FUNCTION_BLOCK "FB_HUB_FW_re"   // FB23, STL
{ S7_Optimized_Access := 'FALSE' }
AUTHOR : MS
// stored: AutoNumber false
   VAR_INPUT
      FW_DBNr : Int;
      SysTime : Time;
   END_VAR
   VAR
      Config : Struct
         Speed : Struct
            Min : Int;   // Mindestgeschwindigkeit in %
            Tipp : Int;   // Geschwindigkeit bei Tipp-Betrieb in %
            Hand : Int;   // maximale Geschwindigkeit bei Hand-Betrieb in %
            Max : Int;   // maximale Geschwindigkeit bei Automatik-Betrieb in %
            Norm : Real;   // Geschwindigkeit in INC/s bei 100%
            endMess : Real;   // gemessene Geschwindigkeit in INC/s bei 100%
         END_STRUCT;
         Rampe : Struct
            Auf_Heben : Real;   // Zeit für Beschleunigung beim Heben von 0% auf 200%
            Ab_Heben : Real;   // Zeit für Verzögerung bei Heben von 200% auf 0%
            Auf_Senken : Real;   // Zeit für Beschleunigung bei Senken von 0% auf 200%
            Ab_Senken : Real;   // Zeit für Verzögerung bei Senken von 200% auf 0%
            NotStop : Real;   // Zeit für Verzögerung bei NotStopp von 200% auf 0%
         END_STRUCT;
         Bereich : Struct
            Pos : DInt;
            Stop : DInt;
            Ziel : DInt;
            Absetzen : DInt;
            Langsam : DInt;
         END_STRUCT;
         TV_Position : DInt;   // Verzögerung Ebenenmitte in ms
         Reaktionszeit : Int;   // Reaktionszeit FU
         Startzeit : Int;   // Zeit Startverzögerung in ms (Zeit von erster Sollwertausgabe bis Istwert>0)
         Variante : Byte;   // Art der Positionierung (0-Absolut, 1-SensorSys, 2-..)
         SimIstSpeed : Byte;   // Variante Simulation Istgeschwindigkeit (0-aus, 1-Soll=Ist,...)
         SimSensors : DWord := DWORD#16#4400_0022;   // Sensoraufbau für Simulation
         SimTakt : DInt;   // Schiebetakt für Sensorsimu in ms
      END_STRUCT;
      IN : Struct
         BA_Tipp : Bool;   // Betriebsart FW Tipp
         BA_Hand : Bool;   // Betriebsart FW Hand
         BA_Auto : Bool;   // Betriebsart FW Auto
         Heben_aktiv : Bool;
         Frg_Hub : Bool;   // Freigabe Positioniervorgang
         Frg_Eil : Bool;   // max. Speed in Automatik und Hand-Speed in Tipp erlaubt
         Break_on : Bool;   // Rückmeldung extern Bremse eingefallen / Hubwerk steht
         mittig : Bool;   // Hub in Posmitte
         resB : Byte;
         HubInc : DInt;   // Istposition in Inkrementen (mm)
         ZielInc : DInt;   // Ziel in Inkrenmenten (mm)
         Absetz_Inc : DInt;   // Inkrement der SU-Ebene des FW
         IstSpeed : Int;   // Istgeschwindigkeit in %
      END_STRUCT;
      OUT : Struct
         Hub_Ok : Bool;   // Positionierung beendet FW steht
         Break_off : Bool;   // Bremse lösen
         res_1 : Bool;
         res_2 : Bool;
         res_3 : Bool;
         res_4 : Bool;
         res_5 : Bool;
         res_6 : Bool;
         resB : Byte;
         Bereich_langsam : DInt;   // berechneter Anhaltebereich
         SollSpeed : Int;   // Sollgeschwindigkeit in %
      END_STRUCT;
      Tmp : Struct
         lastTime : DInt;   // letzter Systemzeitpunkt
         DiffTime : Real;   // Zeit seit letzter Bearbeitung
         lastSpeed : Real;   // letzte ausgegebene Geschwindigkeit
         Messung : Struct
            lastInc : Real;
            addInc : Real;
            addTime : Real;
            lastIst : Int;
            messAct : Bool;
         END_STRUCT;
         StopCount : DInt;
         subInc : Real;
         lastOut : Real;
         TaktCount : Real;   // Taktzähler für Sensorsimu
         PtrSensors : DWord := DWORD#16#0000_0001;
         RunTime : DInt;   // Zeit seit Start Positioniervorgang
      END_STRUCT;
   END_VAR
   VAR_TEMP
      FWDB : Int;
      Rampe_Auf : Real;
      Rampe_Ab : Real;
      minSpeed : Real;
      maxSpeed : Real;
      normSpeed : Real;
      handSpeed : Real;
      TippSpeed : Real;
      IstSpeed : Real;
      Abstand : Real;
      maxDelta : Real;
      Speed : Real;
      tx : Real;
      Rampe_Not : Real;
      incDelta : DInt;
      messAct : Bool;
      posAbsolut : Bool;
      Sensor_on : Bool;
      no_Brms : Bool;
      savD_1 : DInt;
      savD_2 : DInt;
      Korrmax : Real;   // Korrektur max-Speed vom WT
   END_VAR
BEGIN

NETWORK
TITLE = Daten aus FW lesen

      L     #FW_DBNr;
      T     #FWDB;
      OPN   DB [#FWDB];
      AN    "DI_FW_1".IN.Com_Reset;
      JC    nRes;
      L     #SysTime;
      T     #Tmp.lastTime;
      L     0.0;
      T     #Tmp.lastSpeed;
      T     #Tmp.subInc;

nRes: A     "DI_FW_1".ZST.Auto;
      =     #IN.BA_Auto;
      A     "DI_FW_1".ZST.Hand;
      =     #IN.BA_Hand;
      A     "DI_FW_1".ZST.Tipp;
      O     "DI_FW_1".OUT.TIPP;
      =     #IN.BA_Tipp;
      R     #IN.BA_Auto;
      R     #IN.BA_Hand;

      A     "DI_FW_1".OUT.HEBEN_re;
      =     #IN.Heben_aktiv;

      A     "DI_FW_1".OUT.HEBEN_re;
      O     "DI_FW_1".OUT.SENKEN_re;
      =     #IN.Frg_Hub;

      A     "DI_FW_1".OUT.HUB_EIL_re;
      =     #IN.Frg_Eil;

      A     "DI_FW_1".ZST.Mittig;
      =     #IN.mittig;

      A     "DI_FW_1".OUT.no_Brms;
      =     #no_Brms;

      L     "DI_FW_1".HELP.HubInc_re;
      T     #IN.HubInc;
      L     "DI_FW_1".HELP.HubZielInc_re;
      T     #IN.ZielInc;

      L     "DI_FW_1".TMP.low_SU_Ebene;
      L     4;
      *D;
      L     292;
      +D;
      SLD   3;
      LAR1;
      OPN   DB [#FWDB];
      L     DBD [AR1, P#0.0];  //"DI_FW_1".PAR.Hub.Ebene0
      L     #Config.Bereich.Absetzen;
      +D;
      T     #IN.Absetz_Inc;

      L     "DI_FW_1".PAR.Hub.WT_Speed;
      ITD;
      DTR;
      L     100.0;
      /R;
      L     #Config.Speed.Max;
      ITD;
      DTR;
      *R;
      T     #Korrmax;


NETWORK
TITLE = kein Auftrag/Initialisieren
//----------------------------------------
//Positionierart
//----------------------------------------
      L     #Config.Variante;
      L     0;
      ==I;
      =     #posAbsolut;

//----------------------------------------
//Zeitmessung
//----------------------------------------
      L     #SysTime;
      L     #Tmp.lastTime;
      >=D;
      JC    nUms;
      L     16#7FFF_FFFF;  //L#2147483647
      CAC;
      -D;
      L     #SysTime;
      +D;
      JU    Ums;
nUms: -D;
Ums:  DTR;
      T     #Tmp.DiffTime;
      L     10.0;  //Berechnung unter 10ms zu ungenau
      <R;
      BEC;

      L     #SysTime;
      T     #Tmp.lastTime;

//----------------------------------------
//Parametersatz laden
//----------------------------------------
// :::::::::::::::::::::::::::::::::::::::
// Rampen
// :::::::::::::::::::::::::::::::::::::::
      A     #IN.Heben_aktiv;
      O     #IN.BA_Tipp;
      L     #Config.Rampe.Auf_Heben;
      JC    slu;
      L     #Config.Rampe.Auf_Senken;
slu:  L     1000.0;
      *R;
      L     2.0;
      /R;
      T     #Rampe_Auf;

      A     #IN.Heben_aktiv;
      O     #IN.BA_Tipp;
      L     #Config.Rampe.Ab_Heben;
      JC    sld;
      L     #Config.Rampe.Ab_Senken;
sld:  L     1000.0;
      *R;
      L     2.0;
      /R;
      T     #Rampe_Ab;

// :::::::::::::::::::::::::::::::::::::::
// Normalgeschwindigkeit
// :::::::::::::::::::::::::::::::::::::::
      L     #Config.Speed.Norm;
      L     1000.0;
      /R;
      T     #normSpeed;

// :::::::::::::::::::::::::::::::::::::::
// Istgeschwindigkeit
// :::::::::::::::::::::::::::::::::::::::
      L     #IN.IstSpeed;
      ITD;
      DTR;
      ABS;
      L     10000.0;
      /R;
      L     #normSpeed;
      *R;
      T     #IstSpeed;

// :::::::::::::::::::::::::::::::::::::::
// Abstand
// :::::::::::::::::::::::::::::::::::::::
      L     #IN.HubInc;
      L     #IN.ZielInc;
      -D;
      DTR;
      ABS;
      T     #Abstand;

//Korrektur Abstand (Vorhalteweg)um Reaktionszeit auszugleichen
      AN    #posAbsolut;
      JC    StA;
      L     #Config.Reaktionszeit;  //VorhalteWeg=Istspeed * Reaktionszeit
      ITD;  //s = v*t
      DTR;
      L     #IstSpeed;
      *R;
      L     #Abstand;
      CAC;
      -R;
      L     0.0;
      <=R;
      JC    StA;
      CAC;
StA:  T     #Abstand;


// :::::::::::::::::::::::::::::::::::::::
// --- Geschwindigkeiten (Min, Hand, Max)
// :::::::::::::::::::::::::::::::::::::::
      L     #Config.Speed.Tipp;
      A     #IN.BA_Tipp;
      JC    min;
      L     #Config.Speed.Min;
min:  DTR;
      ABS;
      L     100.0;
      /R;
      L     #normSpeed;
      *R;
      T     #minSpeed;

      L     #Config.Speed.Hand;
      DTR;
      ABS;
      L     100.0;
      /R;
      L     #normSpeed;
      *R;
      T     #handSpeed;

      L     #Config.Speed.Tipp;
      DTR;
      ABS;
      L     100.0;
      /R;
      L     #normSpeed;
      *R;
      T     #TippSpeed;

// 2021-07-09 Heben /Senken gleich
      L     #IN.HubInc;
      L     #IN.Absetz_Inc;
      <=D;
      AN    #IN.Frg_Eil;
      A     #IN.mittig;  // Korb am Haken
      O     #IN.BA_Tipp;
      L     #Config.Speed.Tipp;
      JC    max;

      AN    #IN.mittig;
      L     #Config.Speed.Max;  // Höhenwechsel + Freifahren
      JC    max;

      L     #IN.HubInc;
      L     #IN.Absetz_Inc;
      <=D;
      L     #Config.Speed.Hand;
      PUSH;
      +D;
      JC    max;
//
      L     #Config.Speed.Max;
max:  DTR;
      ABS;
      L     #Korrmax;
      >R;
      JC    korr;
      CAC;
korr: L     100.0;
      /R;
      L     #normSpeed;
      *R;
      T     #maxSpeed;
      L     #minSpeed;
      >=R;
      JC    okmx;
      T     #maxSpeed;

//----------------------------------------
//kein Auftrag
//----------------------------------------
okmx: AN    #IN.Frg_Hub;
      JC    Off;

      L     #Tmp.DiffTime;
      L     #Tmp.RunTime;
      +R;
      T     #Tmp.RunTime;

      AN    #IN.BA_Tipp;
      JC    Auto;


NETWORK
TITLE = Tipp
      A     #IN.Frg_Eil;
      L     #maxSpeed;
      JC    Tout;
      L     #minSpeed;
Tout: T     #Speed;
      JU    OutW;

NETWORK
TITLE = Positioniervariante aussuchen
Auto: SET;
      R     #OUT.Hub_Ok;

      L     #Config.Variante;
      JL    vErr;
      JU    vAbs;  //0 Absolut direkt
      JU    vSen;  //1 mit Sensor-System
vErr: JU    Off;


NETWORK
TITLE = Positionierung Absolut direkt
vAbs: NOP   0;

//----------------------------------------
// Bereich_Langsam berechnen
//
// s = (Rampe * Vist * Vist) / (2 * Vnorm)
//----------------------------------------
      L     #Rampe_Ab;
      L     0.0;
      <=R;
      L     #Config.Bereich.Langsam;
      JC    setB;

      L     #IstSpeed;
      SQR;
      L     #Rampe_Ab;
      *R;
      L     #normSpeed;
      /R;
      L     2.0;
      /R;
      RND;
setB: T     #OUT.Bereich_langsam;

//----------------------------------------
// maximal mögl. Geschwindigkeit berechnen
//
// v = SQRT(2 * s * Vnorm / Rampe)
//----------------------------------------
      L     #Abstand;
      L     #Config.Bereich.Ziel;
      DTR;
      >R;
      JC    Sped;

      L     #Abstand;
      L     #Config.Bereich.Stop;
      DTR;
      >R;
      L     #minSpeed;
      JC    setS;

      L     0;
      JU    setS;

Sped: L     #Rampe_Ab;
      L     0.0;
      <=R;
      L     #maxSpeed;
      JC    setS;

      L     2.0;
      L     #Abstand;
      *R;
      L     #normSpeed;
      *R;
      L     #Rampe_Ab;
      /R;
      SQRT;
setS: T     #Speed;

//----------------------------------------
// MAX begrenzen beim Senken (Absetzen)
//
// Vmax = SQRT(2 * Abstand * V100 / t100 + Vhand * Vhand)
//----------------------------------------
      L     #Rampe_Ab;
      L     0.0;
      <=R;
      O     #IN.Heben_aktiv;
      JC    aMax;

      L     #IN.HubInc;
      L     #IN.Absetz_Inc;
      <=D;
      JC    aMax;

      L     #IN.HubInc;
      L     #IN.Absetz_Inc;
      -D;
      DTR;
      L     2.0;
      *R;
      L     #normSpeed;
      *R;
      L     #Rampe_Ab;
      /R;
      L     #handSpeed;
      SQR;
      +R;
      SQRT;
      L     #maxSpeed;
      >R;
      JC    aMax;
      CAC;
      T     #maxSpeed;

//----------------------------------------
// errechnete Geschwindigkeit auf MAX begrenzen
//----------------------------------------
aMax: L     #Speed;
      L     #maxSpeed;
      <=R;
      JC    Ramp;
      T     #Speed;
      JU    Ramp;

//----------------------------------------
// Anstiegsrampe begrenzen
//
// Vdelta = (Vnorm * Tdelta / Rampe)
//----------------------------------------
Ramp: L     #Speed;
      L     #IstSpeed;
      <=R;
      JC    aMin;

      L     #Rampe_Auf;
      L     0.0;
      <=R;
      JC    aMin;

      L     #Tmp.RunTime;
      L     #Config.Startzeit;
      DTR;
      <R;
      L     #minSpeed;
      JC    altw;

      L     #normSpeed;
      L     #Tmp.DiffTime;
      *R;
      L     #Rampe_Auf;
      /R;
      T     #maxDelta;

      L     #Speed;
      L     #Tmp.lastOut;
      -R;
      ABS;
      L     #maxDelta;
      <=R;
      JC    aMin;

      L     #Tmp.lastOut;
      +R;
altw: T     #Speed;

//----------------------------------------
// errechnete Geschwindigkeit auf MIN begrenzen
//----------------------------------------
aMin: L     #Speed;
      L     #minSpeed;
      >=R;
      JC    Out;

      T     #Speed;

      JU    Out;


NETWORK
TITLE = Positionierung mit Sensor-System
vSen: SET;
// -------------------------------
// Geschwindigkeit berechnen
// -------------------------------
      L     #Abstand;
      L     #Config.Bereich.Langsam;
      DTR;
      >R;
      L     #maxSpeed;
      JC    vSet;

      L     #Abstand;
      L     #Config.Bereich.Ziel;
      DTR;
      <=R;
      L     #minSpeed;
      JC    vSet;

      A     #no_Brms;
      L     #maxSpeed;
      JC    vSet;

      L     #handSpeed;
      L     #maxSpeed;
      >R;
      JC    vSet;
      CAC;

vSet: T     #Speed;

// -------------------------------
// Rampen begrenzen
// -------------------------------
      L     #Speed;
      L     #IstSpeed;
      >R;
      JC    rAuf;
      <R;
      JC    rAb;
      JU    Out;

rAuf: L     0.0;
      L     #Rampe_Auf;
      >=R;
      JC    Out;

      L     #Tmp.RunTime;
      L     #Config.Startzeit;
      DTR;
      >=R;
      JC    wtr2;

      L     #minSpeed;
      JU    outS;

wtr2: L     #normSpeed;
      L     #Tmp.DiffTime;
      *R;
      L     #Rampe_Auf;
      /R;
      T     #maxDelta;

      L     #Speed;
      L     #Tmp.lastOut;
      -R;
      ABS;
      L     #maxDelta;
      <=R;
      JC    Out;

      L     #Tmp.lastOut;
      +R;
outS: T     #Speed;
      JU    Out;

rAb:  L     0.0;
      L     #Rampe_Ab;
      >=R;
      JC    Out;

      L     #normSpeed;
      L     #Tmp.DiffTime;
      *R;
      L     #Rampe_Ab;
      /R;
      T     #maxDelta;

      L     #Tmp.lastOut;
      L     #Speed;
      -R;
      ABS;
      L     #maxDelta;
      <=R;
      JC    Out;

      L     #Tmp.lastOut;
      CAC;
      -R;
      T     #Speed;
      JU    Out;


NETWORK
TITLE = Ausgabe
Out:  L     #Abstand;
      L     #Config.Bereich.Ziel;
      DTR;
      >R;
      L     #Config.TV_Position;
      DTR;
      JC    setT;

      L     #minSpeed;
      T     #Speed;

      L     #Tmp.StopCount;
      L     0.0;
      <=R;
      O(;
      L     #Abstand;
      L     #Config.Bereich.Stop;
      DTR;
      <=R;
      A     #posAbsolut;
      );
      JC    Off;

      L     #Tmp.StopCount;
      L     #Tmp.DiffTime;
      -R;

setT: T     #Tmp.StopCount;
      JU    OutW;

Off:  A     #IN.Break_on;
      S     #OUT.Hub_Ok;

      L     0;
      T     #OUT.Bereich_langsam;
      L     0.0;
      T     #Speed;
      T     #Tmp.lastOut;
      T     #Tmp.RunTime;
      JU    OutW;

OutW: L     #Speed;
      T     #Tmp.lastOut;
      L     100.0;
      *R;
      L     #normSpeed;
      /R;
      T     #maxDelta;
      TRUNC;
      T     #OUT.SollSpeed;

      L     #Tmp.RunTime;
      L     #Config.Startzeit;
      DTR;
      >=R;
      A     #IN.Frg_Hub;
      S     #OUT.Break_off;

      L     #OUT.SollSpeed;
      L     0;
      ==I;
      ON    #IN.Frg_Hub;
      R     #OUT.Break_off;


NETWORK
TITLE = Messung der Normgeschwindigkeit
      L     #IN.IstSpeed;
      L     #Tmp.Messung.lastIst;
      -I;
      JP    cNeg;
      NEGI;
cNeg: L     100;
      <=I;
      A     #IN.Frg_Hub;
      =     #messAct;
      JC    cOn;
//----------------------------------------
// Messung aus
// Werte initialisieren
//----------------------------------------
      L     0.0;
      T     #Tmp.Messung.addTime;
      T     #Tmp.Messung.addInc;

      L     #IN.IstSpeed;
      T     #Tmp.Messung.lastIst;
      JU    cEnd;

//----------------------------------------
// Messung läuft
// Werte aufzeichnen
//----------------------------------------
cOn:  L     #IN.HubInc;
      DTR;
      L     #Tmp.Messung.lastInc;
      -R;
      ABS;
      L     #Tmp.Messung.addInc;
      +R;
      T     #Tmp.Messung.addInc;

      L     #Tmp.DiffTime;
      L     #Tmp.Messung.addTime;
      +R;
      T     #Tmp.Messung.addTime;

//----------------------------------------
// Messung läuft lange genug
// um Werte zu berechnen
//----------------------------------------
      L     #Tmp.Messung.addTime;
      L     1000.0;
      <R;
      JC    cEnd;
      /R;
      L     #Tmp.Messung.addInc;
      CAC;
      /R;
      L     #Tmp.Messung.lastIst;
      ITD;
      DTR;
      ABS;
      /R;
      L     10000.0;
      *R;
      T     #Config.Speed.endMess;
      JU    cEnd;

cEnd: L     #IN.HubInc;
      DTR;
      T     #Tmp.Messung.lastInc;



NETWORK
TITLE = Daten in FW schreiben

      OPN   DB [#FWDB];

      A     #OUT.Hub_Ok;
      =     "DI_FW_1".IN.Hub_ok_re;

      L     #OUT.SollSpeed;
      T     "DI_FW_1".HELP.Speed_Hub_re;


NETWORK
TITLE = Simulation Ist-Wert-Rückgabe
      L     #Config.SimIstSpeed;
      L     0;
      ==I;
      JC    simu;

      L     #OUT.SollSpeed;
      T     #IN.IstSpeed;

simu: NOP   0;


NETWORK
TITLE = Simulation Bewegung
      AN    "DB_ANLAGE".BA.Simulation;
      BEC;

      AN    #OUT.Break_off;
      =     #IN.Break_on;

      A     #IN.Heben_aktiv;
      JC    sTra;
      L     #Speed;
      NEGR;
      T     #Speed;
sTra: L     #Config.Rampe.NotStop;
      L     0.0;
      <=R;
      JC    Ink;

      L     #Config.Rampe.NotStop;
      L     1000.0;
      *R;
      L     2.0;
      /R;
      T     #Rampe_Not;

      L     #normSpeed;
      L     #Tmp.DiffTime;
      *R;
      L     #Rampe_Not;
      /R;
      T     #maxDelta;

      L     #Speed;
      L     #Tmp.lastSpeed;
      -R;
      ABS;
      L     #maxDelta;
      <=R;
      JC    Ink;

      L     #Speed;
      L     #Tmp.lastSpeed;
      <R;
      L     #Tmp.lastSpeed;
      L     #maxDelta;
      JC    sub;
      +R;
      JU    stt;
sub:  -R;
stt:  T     #Speed;

Ink:  L     #Config.Variante;
      JL    sErr;
      JU    sAbs;  //0 Absolut direkt
      JU    sSen;  //1 mit Sensor-System
sErr: JU    OutS_Mig;

//----------------------------------------
// Simu Absolut
//----------------------------------------
sAbs: L     #Speed;
      L     #Tmp.lastSpeed;
      +R;
      L     2.0;
      /R;
      L     #Tmp.DiffTime;
      *R;
      L     #Tmp.subInc;
      +R;
      T     #Tmp.subInc;

      TRUNC;
      T     #incDelta;
      L     #IN.HubInc;  // init startinkrement
      +D;
      OPN   DB [#FWDB];
      T     "DI_FW_1".HELP.HubInc_re;

      L     #Tmp.subInc;
      L     #incDelta;
      DTR;
      -R;
      T     #Tmp.subInc;
      JU    OutS_Mig;

//------------------------------------------
// Simu Sensoren
//------------------------------------------

// :::::::::::::::::::::::::::::::::::::::::
// Simulationstakt entsprechend IstSpeed
// verlängern oder verkürzen
// :::::::::::::::::::::::::::::::::::::::::
sSen: L     #Speed;
      L     #Tmp.lastSpeed;
      +R;
      L     2.0;
      /R;
      ABS;
      L     #normSpeed;
      /R;
      L     #Tmp.DiffTime;
      *R;
      L     #Tmp.TaktCount;
      CAC;
      -R;
      T     #Tmp.TaktCount;

// :::::::::::::::::::::::::::::::::::::::::
// Simutakt abgelaufen --> Pointer schieben
// :::::::::::::::::::::::::::::::::::::::::
      L     0.0;
      L     #Tmp.TaktCount;
      <R;
      ON    #IN.Frg_Hub;
      JC    sInc;
      L     #Config.SimTakt;
      DTR;
      +R;
      T     #Tmp.TaktCount;

      L     0;
      L     #Tmp.PtrSensors;
      ==D;
      JC    UIn;

      L     #Tmp.PtrSensors;  //Pointer (virtuelle Höhe)
      A     #IN.Heben_aktiv;
      JC    hSim;
      SRD   1;  //Pointer (virtuelle Höhe) nach unten
      JP    UIn;  //Unterlauf
      JU    tSim;
hSim: SLD   1;  //Pointer (virtuelle Höhe) nach oben
      JP    OIn;  //Überlauf
tSim: T     #Tmp.PtrSensors;

// :::::::::::::::::::::::::::::::::::::::::
// Istposition ermitteln
// :::::::::::::::::::::::::::::::::::::::::
sInc: L     0;
      T     #incDelta;
      SET;
      R     #Sensor_on;

      L     #Tmp.PtrSensors;  //Zeiger auf virtuelle Höhe
      L     #Config.SimSensors;  //Jedes Bit=1 ist ein Sensor
retR: SRD   1;  //nach Sensoren suchen
      JP    posR;

      A     #Sensor_on;  //Sensor verlassen --> Zählen
      R     #Sensor_on;
      JC    cntR;
      JU    nexR;

posR: AN    #Sensor_on;  //Sensor erreicht --> Zählen
      S     #Sensor_on;
      JC    cntR;
      JU    nexR;

cntR: T     #savD_1;  //Akku 1 retten
      CAC;
      T     #savD_2;  //Akku 2 retten
      L     #incDelta;  //Inkrement erhöhen
      L     1;
      +D;
      T     #incDelta;
      L     #savD_2;  //Akkus wieder herstellen
      L     #savD_1;  //geschobene Werte zur weiterverarbeitung

nexR: CAC;
      SRD   1;  //Pointer schieben
      JP    endR;  //Pointer gefunden --> alle Inkremente gezählt
      CAC;
      JU    retR;  //weiterzählen

endR: L     #incDelta;
      OPN   DB [#FWDB];
      T     %DBD8;  //"DI_FW_1".ZST.HubInc
      JU    OutS_Mig;

UIn:  L     1;  //bei Unterlauf Pointer initialisieren
      T     #Tmp.PtrSensors;
      JU    OutS_Mig;

OIn:  L     16#8000_0000;  //bei Überlauf Pointer initialisieren
      T     #Tmp.PtrSensors;
      JU    OutS_Mig;

//----------------------------------------
// Ausgabe Geschwindigkeit
//----------------------------------------
OutS_Mig:L     #Speed;
      T     #Tmp.lastSpeed;


      L     #Config.SimIstSpeed;
      L     0;
      <>I;
      BEC;

      L     #Tmp.lastSpeed;
      L     10000.0;
      *R;
      L     #normSpeed;
      /R;
      ABS;
      TRUNC;
      T     #IN.IstSpeed;

END_FUNCTION_BLOCK

FUNCTION "FC_FW_SCHIEBEN" : Void   // FC21, STL
{ S7_Optimized_Access := 'FALSE' }
AUTHOR : MS
// stored: AutoNumber false
   VAR_TEMP
      count_FW : Byte;
      FW_DB_1 : Word;
      FW_DB_2 : Word;
      QT_DB : Word;
      CHK_POS_min : Int;
      CHK_POS_max : Int;
      CHK_Z_min : DInt;
      CHK_Z_max : DInt;
      CHK_POS : Int;
      CHK_Z : Int;
      PosFW : DInt;
      SchiebePos : DInt;
      SchiePos : Byte;
      schieben : Bool;
      count : Int;
      Rcount : Byte;   // Reihenzähler QT
      ZielBereich : DInt;
      Schwerpunkt : Byte;
      ziel : Int;
      FW_Nr : Int;
      erlaubt : Bool;
      Offset : Bool;
   END_VAR
BEGIN

NETWORK
TITLE = 
      L     "DB_ANLAGE".config.ANZ_FW;
      L     1;
      -I;
      T     #count_FW;
ret:  L     #count_FW;
      L     0;
      <=I;
      JC    NW3;

      L     #count_FW;
      L     10;
      +I;
      T     #FW_DB_1;
      L     1;
      +I;
      T     #FW_DB_2;

//------------------------
//SCHIEBEMERKER RESET
//------------------------
      OPN   DB [#FW_DB_1];
      L     %DBW30;  //Liegt Befehl an ?
      L     0;
      ==I;
      A     %DBX13.0;  //"DI_FW_1".ZST.schieben
      R     %DBX13.0;  //"DI_FW_1".ZST.schieben

      OPN   DB [#FW_DB_2];
      L     %DBW30;  //Liegt Befehl an ?
      L     0;
      ==I;
      A     %DBX13.0;  //"DI_FW_2".ZST.schieben
      R     %DBX13.0;  //"DI_FW_2".ZST.schieben

//------------------------
//FW rückwärts schieben
//------------------------
      OPN   DB [#FW_DB_1];

      AN    %DBX1.6;  //"DBI_FW_1".ZST.Auto
      AN    %DBX1.5;  //"DBI_FW_1".ZST.Auto_Stop
      AN(;
      A     %DBX1.4;  //"DI_FW_1".ZST.Hand
      A     %DBX13.5;  //"DI_FW_1".ZST.schieben_erlaubt
      );
      ON    %DBX0.0;  //"DBI_FW_1".ZST.BEREIT
      O     %DBX0.1;  //aktiv
      O     %DBX0.2;  //Fehler
      O     %DBX13.0;  //"DI_FW_1".ZST.schieben
      JC    NW2;

      OPN   DB [#FW_DB_2];  //keine bzw. andere Fahrtrichtung
      L     0;
      L     %DBB351;  //"DI_FW_2".TMP.ZielPos
      ==I;
      ON    %DBX0.7;  //"DBI_FW_2".ZST.RUECKWAERTS_AKT
      JC    NW2;

      L     %DBB351;  //"DI_FW_2".TMP.ZielPos
      L     "DB_POS".LENG;
      *I;
      L     "DB_POS".Offset;
      +I;
      SLD   3;
      LAR1;
      OPN   "DB_POS";
      L     DBD [AR1, P#22.0];  //Position des Zielbades in Inkrementen
      OPN   DB [#FW_DB_1];
      L     %DBD198;  //"DI_FW_1".PAR.Fahrt.Abstand_vor
      -D;
//      L     DBW  234                    //"DI_FW_1".PAR.Fahrt.SoftOffset
//      -D
      OPN   DB [#FW_DB_2];
      L     %DBD212;  //"DI_FW_2".PAR.Fahrt.Bereich_Pos
      -D;
      T     #SchiebePos;
      OPN   DB [#FW_DB_1];
      L     %DBD4;  //"DI_FW_1".ZST.PosInc
      >=D;
      JC    NW2;
      OPN   DB [#FW_DB_1];
      L     #SchiebePos;
      L     %DBD212;  //"DI_FW_1".PAR.Fahrt.Bereich_Pos
      -D;
      T     #SchiebePos;

      L     0;
      L     %DBW396;  //"DI_FW_1".TMP.nexQuelle
      ==I;
      JC    noRe;
      L     "DB_POS".LENG;
      *I;
      L     "DB_POS".Offset;
      +I;
      SLD   3;
      LAR1;
      OPN   "DB_POS";
      L     #SchiebePos;
      L     DBD [AR1, P#22.0];  //Position des Zielbades in Inkrementen
      >=D;
      JC    NW2;

noRe: OPN   DB [#FW_DB_1];
      L     %DBB2;  //"DBI_FW_1".ZST.POSITION
retR: T     #count;
      OPN   DB [#FW_DB_1];
      L     %DBB194;  //"DI_FW_1".PAR.Fahrt.FAHRBEREICH_MIN
      <I;
      JC    NW2;

      L     #count;
      L     "DB_POS".LENG;
      *I;
      L     "DB_POS".Offset;
      +I;
      SLD   3;
      LAR1;
      OPN   "DB_POS";
      L     #SchiebePos;
      L     DBD [AR1, P#22.0];  //BadPosition
      >=D;
      JC    TakR;

      L     #count;
      L     1;
      -I;
      JU    retR;

TakR: OPN   DB [#FW_DB_1];
      S     %DBX13.0;  //"DI_FW_1".ZST.schieben
      L     16#FF01;
      T     %DBW30;  //Befehlskennung
      L     #count;
      T     %DBB32;  //FW Ziel
      L     #SchiebePos;
      T     %DBD38;  //"DI_FW_1".ZST.SchiebeInc


NETWORK
TITLE = 
//------------------------
//FW vorwärts schieben
//------------------------
NW2:  OPN   DB [#FW_DB_2];
      AN    %DBX1.6;  //"DBI_FW_2".ZST.Auto
      AN    %DBX1.5;  //"DBI_FW_2".ZST.Auto_Stop
      AN    %DBX1.4;  //"DI_FW_2".ZST.Hand
      ON    %DBX13.5;  //"DI_FW_2".ZST.schieben_erlaubt
      ON    %DBX0.0;  //"DBI_FW_2".ZST.BEREIT
      O     %DBX0.1;  //aktiv
      O     %DBX0.2;  //Fehler
      O     %DBX13.0;  //"DI_FW_2".ZST.schieben
      JC    nxt;

      OPN   DB [#FW_DB_1];
      L     0;
      L     %DBB351;  //"DI_FW_1".TMP.ZielPos
      ==I;
      ON    %DBX0.6;  //"DBI_FW_1".ZST.VORWAERTS_AKT
      JC    nxt;

      L     %DBB351;  //"DI_FW_1".TMP.ZielPos
      L     "DB_POS".LENG;
      *I;
      L     "DB_POS".Offset;
      +I;
      SLD   3;
      LAR1;
      OPN   "DB_POS";
      L     DBD [AR1, P#22.0];  //Position des Zielbades in Inkrementen
      OPN   DB [#FW_DB_1];
      L     %DBD198;  //"DI_FW_1".PAR.Fahrt.Abstand_vor
      +D;
//      L     DBW  234                    //"DI_FW_1".PAR.Fahrt.SoftOffset
//      +D
      OPN   DB [#FW_DB_2];
      L     %DBD212;  //"DI_FW_2".PAR.Fahrt.Bereich_Pos
      +D;
      T     #SchiebePos;
      L     %DBD4;  //"DI_FW_2".ZST.PosInc
      <=D;
      JC    nxt;
      OPN   DB [#FW_DB_1];
      L     #SchiebePos;
      L     %DBD212;  //"DI_FW_1".PAR.Fahrt.Bereich_Pos
      +D;
      T     #SchiebePos;

      OPN   DB [#FW_DB_2];
      L     0;
      L     %DBW396;  //"DI_FW_1".TMP.nexQuelle
      ==I;
      JC    noLi;
      L     "DB_POS".LENG;
      *I;
      L     "DB_POS".Offset;
      +I;
      SLD   3;
      LAR1;
      OPN   "DB_POS";
      L     #SchiebePos;
      L     DBD [AR1, P#22.0];  //Position des Zielbades in Inkrementen
      <=D;
      JC    nxt;

noLi: OPN   DB [#FW_DB_2];
      L     %DBB2;  //"DBI_FW_2".ZST.POSITION
retV: T     #count;
      OPN   DB [#FW_DB_2];
      L     %DBB195;  //"DI_FW_2".PAR.Fahrt.FAHRBEREICH_MAX
      >I;
      JC    nxt;

      L     #count;
      L     "DB_POS".LENG;
      *I;
      L     "DB_POS".Offset;
      +I;
      SLD   3;
      LAR1;
      OPN   "DB_POS";
      L     #SchiebePos;
      L     DBD [AR1, P#22.0];  //BadPosition
      <=D;
      JC    TakL;

      L     #count;
      L     1;
      +I;
      JU    retV;

TakL: OPN   DB [#FW_DB_2];
      S     %DBX13.0;  //"DI_FW_2".ZST.schieben
      L     16#FF01;
      T     %DBW30;  //Befehlskennung
      L     #count;
      T     %DBB32;  //FW Ziel
      L     #SchiebePos;
      T     %DBD38;  //"DI_FW_1".ZST.SchiebeInc

nxt:  L     #count_FW;
      DEC   1;
      T     #count_FW;
      JU    ret;


NETWORK
TITLE = QT schiebt FW
NW3:  NOP   0;

      L     0;
      T     #SchiebePos;

//Es gibt keine QT
      L     0;
      L     "DB_ANLAGE".config.ANZ_QT;
      >=I;
      BEC;

//QT Prüfschleife

      L     30;
      +I;
reQ:  T     #QT_DB;

      OPN   DB [#QT_DB];
      L     %DBB104;  //"DBI_QT_1".TMP.ZIEL_REIHE QT will nicht fahren
      L     0;
      ==I;
      O(;
      L     %DBB100;  //"DI_QT_1".TMP.ZIEL_POS
      L     0;
      ==I;
      );
      JC    nxtQ;

//Ermittlung gesperrter Bereich um QT-Zielposition
      OPN   DB [#QT_DB];
      L     0;
      T     #Rcount;

reR:  L     #Rcount;
      L     5;
      >=I;
      JC    nxtQ;

      OPN   DB [#QT_DB];
      L     #Rcount;
      L     60;
      +D;
      SLD   3;
      LAR1;

      L     0;
      L     DBB [AR1, P#0.0];  //"DBI_QT_1".PAR.POS1..5
      ==I;
      JC    nxtQ;
      T     #CHK_POS;

      L     "DB_POS".LENG;
      *I;
      L     "DB_POS".Offset;
      +I;
      SLD   3;
      LAR1;
      OPN   "DB_POS";
      L     DBD [AR1, P#22.0];  //BadPosition
      L     DBW [AR1, P#26.0];  //Abstand_vor
      +D;
      T     #CHK_Z_max;

      L     DBD [AR1, P#22.0];  //BadPosition
      L     DBW [AR1, P#28.0];  //Abstand_rck
      -D;
      T     #CHK_Z_min;

      L     DBB [AR1, P#3.0];  //Schiebepos
      T     #SchiePos;

      L     "DB_ANLAGE".config.ANZ_FW;
      L     10;
      +I;
reF:  T     #FW_DB_1;

      OPN   DB [#FW_DB_1];
      AN    %DBX1.6;  //"DBI_FW_1".ZST.Auto
      AN    %DBX1.5;  //"DBI_FW_1".ZST.Auto_Stop
//  UN    DBX    1.4                  //"DI_FW_2".ZST.Hand
      ON    %DBX13.5;  //"DI_FW_2".ZST.schieben_erlaubt
      ON    %DBX0.0;  //"DBI_FW_1".ZST.BEREIT
      O     %DBX0.1;  //aktiv
      O     %DBX0.2;  //Fehler
      O     %DBX13.0;  //"DI_FW_1".ZST.schieben
      JC    nxtF;
      R     #schieben;

      OPN   DB [#FW_DB_1];
      L     %DBD4;  //"DI_FW_1".ZST.PosInc
      T     #PosFW;
      L     %DBD220;  //"DI_FW_1".PAR.Fahrt.Bereich_Ziel
      T     #ZielBereich;

//      L     #CHK_Z_max
//      L     #ZielBereich
//      +D
//      T     #CHK_Z_max

      L     #PosFW;
      L     #CHK_Z_max;
      >=D;
      JC    nxtF;

//      L     #CHK_Z_min
//      L     #ZielBereich
//      -D
//      T     #CHK_Z_min

      L     #PosFW;
      L     #CHK_Z_min;
      <=D;
      JC    nxtF;
      S     #schieben;

      AN    #schieben;
      JC    nxtF;

      L     #CHK_Z_max;
      L     #ZielBereich;
      +D;
      T     #CHK_Z_max;

      L     #CHK_Z_min;
      L     #ZielBereich;
      -D;
      T     #CHK_Z_min;

      L     0;
      L     #SchiePos;  //keine Schiebepos definiert
      ==I;  //deshalb in Richtung Schwerpunkt schieben
      =     #Offset;
      JC    such;

fnd:  L     #SchiePos;
      T     #ziel;
      L     0;
      ==I;
      JC    nxtF;

      OPN   DB [#FW_DB_1];
      L     0;
      L     %DBW396;  //"DI_FW_1".TMP.nexQuelle
      ==I;
      JC    noQ;
      L     "DB_POS".LENG;
      *I;
      L     "DB_POS".Offset;
      +I;
      SLD   3;
      LAR1;
      OPN   "DB_POS";
      L     #CHK_Z_min;
      L     DBD [AR1, P#22.0];  //Position des Zielbades in Inkrementen
      <=D;
      O(;
      L     #CHK_Z_max;
      L     DBD [AR1, P#22.0];  //Position des Zielbades in Inkrementen
      >=D;
      );
      JC    nxtF;

noQ:  L     #FW_DB_1;
      +     -10;
      T     #FW_Nr;

      CALL  "FC_FW_Befehl_ok"
      ( FW_Nr    := #FW_Nr,
        kl_Z     := #ziel,
        Gr_Z     := #ziel,
        QT_Check := FALSE,
        Ablassen := FALSE,
        vor      := FALSE,
        chk_on   := FALSE,
        erlaubt  := #erlaubt
      );

      AN    #erlaubt;
      JC    nxtF;

      OPN   DB [#FW_DB_1];
      L     16#F001;
      AN    #Offset;
      JC    toPo;
      L     16#FF01;
toPo: T     %DBW30;  //Befehlskennung
      L     #SchiePos;
      T     %DBB32;  //FW Ziel
      L     #SchiebePos;
      T     %DBD38;  //"DI_FW_1".ZST.SchiebeInc

nxtF: L     #FW_DB_1;
      L     11;
      <=I;
      JC    nxR;

      L     #FW_DB_1;
      L     1;
      -I;
      T     #FW_DB_1;
      JU    reF;

nxtQ: L     #QT_DB;
      L     31;
      <=I;
      BEC;

      L     #QT_DB;
      L     1;
      -I;
      JU    reQ;

nxR:  L     #Rcount;
      L     1;
      +I;
      T     #Rcount;
      JU    reR;

//Suche nach Schiebepos in Richtung Schwerpunkt
such: L     #CHK_POS;
      T     #SchiePos;

      OPN   DB [#FW_DB_1];
      L     0;
      L     %DBW396;  //"DI_FW_1".TMP.nexQuelle
      ==I;
      JC    spnt;
      JU    pkt;

spnt: OPN   DB [#FW_DB_1];
      L     %DBB194;  //"DI_FW_1".PAR.Fahrt.FAHRBEREICH_MIN
      L     %DBB195;  //"DI_FW_1".PAR.Fahrt.FAHRBEREICH_MAX
      +I;
      L     2;
      /I;
pkt:  T     #Schwerpunkt;

      L     #CHK_POS;
      L     #Schwerpunkt;
      >=I;
      JC    Srck;  //Schiebe rückwärts

Svor: L     #SchiePos;
      L     1;
      +I;
      T     #SchiePos;

      L     "DB_POS".LENG;
      *I;
      L     "DB_POS".Offset;
      +I;
      SLD   3;
      LAR1;
      OPN   "DB_POS";
      L     DBD [AR1, P#22.0];  //BadPosition
      L     #CHK_Z_max;
      <D;
      JC    Svor;
      T     #SchiebePos;
      JU    fnd;

Srck: L     #SchiePos;
      L     1;
      -I;
      T     #SchiePos;

      L     "DB_POS".LENG;
      *I;
      L     "DB_POS".Offset;
      +I;
      SLD   3;
      LAR1;
      OPN   "DB_POS";
      L     DBD [AR1, P#22.0];  //BadPosition
      L     #CHK_Z_min;
      >D;
      JC    Srck;
      T     #SchiebePos;
      JU    fnd;

END_FUNCTION

FUNCTION "FC_FW_Befehl_ok" : Void   // FC20, STL
TITLE = Prüfung ob Befehl ausführbar
{ S7_Optimized_Access := 'FALSE' }
AUTHOR : MS
// stored: AutoNumber false
   VAR_INPUT
      FW_Nr : Int;
      kl_Z : Int;
      Gr_Z : Int;
      QT_Check : Bool;
      Ablassen : Bool;   // Tropfschale ablassen anfahren mit Posversatz
      vor : Bool;   // Bewegung vorwärts --> Quelle < Ziel
      chk_on : Bool;
   END_VAR
   VAR_OUTPUT
      erlaubt : Bool;
   END_VAR
   VAR_TEMP
      Save_AR1 : DWord;
      Save_AR2 : DWord;
      ZielInc : DInt;
      IstInc : DInt;
      PosmitteInc : DInt;   // Inkrement der Positionsmitte
      PosBereich : DInt;   // Bereich um Positionsmitte
      FW_DB : Int;
      Quelle : Int;
      Ziel : Int;
      aktZiel : Int;
      temp_kl_Z : Int;
      temp_Gr_Z : Int;
      Row : Byte;   // Reihe, welche zu prüfen ist
      FW_count : Byte;
      IstPos : Byte;
      nRowChk : Bool;   // Reihe nicht prüfen
      low_FW : Bool;
      high_FW : Bool;
      vor_akt : Bool;
      rck_akt : Bool;
      Q_null : Bool;
      TW_in_Quelle : Bool;
      temp_erlaubt : Bool;
   END_VAR
BEGIN

NETWORK
TITLE = Initialisierung
//Adressregister retten
      TAR1;
      T     #Save_AR1;
      TAR2;
      T     #Save_AR2;

// init
      SET;
      S     #temp_erlaubt;

      L     #FW_Nr;
      L     1;
      ==I;
      =     #low_FW;
      CAC;
      L     "DB_ANLAGE".config.ANZ_FW;
      ==I;
      =     #high_FW;

      L     #kl_Z;
      T     #temp_kl_Z;

      L     #Gr_Z;
      T     #temp_Gr_Z;

NETWORK
TITLE = nach links (zum niedrigeren) suchen
//Es existiert links kein FW
      A     #low_FW;
      JC    sre;

//-----------------------------------------
//kleinstes Ziel PosInc laden
      L     #temp_kl_Z;
      L     "DB_POS".LENG;
      *I;
      L     "DB_POS".Offset;
      +I;
      SLD   3;
      LAR1;
      OPN   "DB_POS";
      L     DBD [AR1, P#22.0];  //BadPos in Inkrementen
      T     #PosmitteInc;
      AN    #Ablassen;
      JC    nab1;
      L     DBD [AR1, P#64.0];  //"DB_POS".POS[0].SonderPos_Offset
      +D;
nab1: T     #ZielInc;
//-----------------------------------------

//-----------------------------------------
//Start-FW laden
      L     #FW_Nr;
      T     #FW_count;
      L     10;
      +I;
      T     #FW_DB;

      OPN   DB [#FW_DB];
      L     #ZielInc;
      L     %DBD212;  //"DI_FW_1".PAR.Fahrt.Bereich_Pos
      -D;
      T     #ZielInc;

      OPN   DB [#FW_DB];
      L     %DBB186;  //"DI_FW_1".PAR.Reihe
      T     #Row;
      L     0;
      ==I;
      =     #nRowChk;

      OPN   DB [#FW_DB];
      L     %DBB2;  //"DI_FW_1".ZST.POSITION
      T     #IstPos;
      L     %DBD4;  //"DI_FW_1".ZST.PosInc
      T     #IstInc;
      L     %DBD212;  //"DI_FW_1".PAR.Fahrt.Bereich_Pos
      T     #PosBereich;
//-----------------------------------------

//-----------------------------------------
//Bewegt sich der zu prüfende TW
//immer in Richtung größere Position
      L     #PosmitteInc;
      L     #PosBereich;
      +D;
      L     #IstInc;
      >=D;
      A(;
      L     #IstPos;
      L     #temp_kl_Z;
      <=I;
      );
      AN(;
      L     #temp_kl_Z;
      L     #temp_Gr_Z;
      ==I;
      );
      A     #vor;
      A     #chk_on;
      JC    sre;
//-----------------------------------------

//-----------------------------------------
//Nachbar-FW prüfen
retl: L     #FW_count;
      +     -1;
      T     #FW_count;
      L     1;
      <I;
      JC    sre;

      L     #FW_count;
      L     10;
      +I;
      T     #FW_DB;
      OPN   DB [#FW_DB];
//-----------------------------------------

//-----------------------------------------
//Reihe prüfen
      A     #nRowChk;
      JC    nRl;
      L     0;
      L     %DBB186;  //"DI_FW_1".PAR.Reihe
      ==I;
      S     #nRowChk;
      JC    nRl;
      L     #Row;  //Ende der Reihe
      <>I;
      JC    sre;
//-----------------------------------------

//-----------------------------------------
//Zielinkrement korrigieren
nRl:  L     #ZielInc;
      L     %DBD198;  //"DI_FW_2".PAR.Fahrt.Abstand_vor
      -D;
      L     %DBD212;  //"DI_FW_1".PAR.Fahrt.Bereich_Pos
      -D;
      T     #ZielInc;
//-----------------------------------------

//-----------------------------------------
//Quelle/Ziel prüfen
      L     %DBB32;
      T     #Quelle;
      L     %DBB33;
      T     #Ziel;
      L     %DBB351;  //"DI_FW_1".TMP.ZielPos
      T     #aktZiel;
      A     %DBX0.7;  //"DI_FW_1".ZST.RUECKWAERTS_AKT
      =     #rck_akt;

      L     #Ziel;
      L     0;
      ==I;
      A(;
      L     #Quelle;
      <>I;
      );
      JCN   okl;
      T     #Ziel;
      L     0;
      T     #Quelle;
//-----------------------------------------

//-----------------------------------------
//FW muss geschoben werden
okl:  L     #Quelle;
      L     #Ziel;
      +I;
      L     0;
      ==I;
      O(;
      L     #aktZiel;
      L     #Ziel;
      ==I;
      A(;
      L     %DBB2;  //"DI_FW_1".ZST.POSITION
      ==I;
      A     %DBX53.2;  //"DI_FW_1".IN.Pos_ok
      AN    %DBX0.6;  //"DI_FW_1".ZST.VORWAERTS_AKT
      );
      );
      =     #TW_in_Quelle;
      JC    sRe_Mig;

//neu Test Nachfahren
      L     #Quelle;
      L     0;
      ==I;
      =     #Q_null;

      L     #Quelle;
      L     #Ziel;
      ==I;
      AN    #TW_in_Quelle;
      JC    sRe_Mig;

      L     #aktZiel;
      L     #Ziel;
      ==I;
      A(;
      L     #Quelle;
      <=I;
      AN    #Q_null;
      O(;
      A     #Q_null;
      A     #rck_akt;
      );
      );
      JC    sRe_Mig;
      JU    nSRe;

sRe_Mig:L     #temp_kl_Z;
rpol: T     #Quelle;
      L     1;
      <I;
      R     #temp_erlaubt;
      JC    ende;

      L     #Quelle;
      L     "DB_POS".LENG;
      *I;
      L     "DB_POS".Offset;
      +I;
      SLD   3;
      LAR1;
      OPN   "DB_POS";
//Reihe zu ende?
      A     #nRowChk;
      JC    spol;
      L     DBB [AR1, P#4.0];  //"DB_POS".POS[0].Reihe
      L     #Row;
      <>I;
      R     #temp_erlaubt;
      JC    ende;

//mögliche Schiebepos?
spol: L     #ZielInc;
      L     DBD [AR1, P#22.0];  //BadPos in Inkrementen
      <D;
      JC    nxQl;
      T     #ZielInc;
      JU    retl;

nxQl: L     #Quelle;
      +     -1;
      JU    rpol;
//-----------------------------------------

//-----------------------------------------
nSRe: L     0;
      L     #Ziel;
      ==I;
      JC    tstl;  //Leerfahrt- oder Schiebebefehl
      L     #aktZiel;
      ==I;
      JC    chkl;  //Quelle bereits bedient
tstl: L     #Quelle;
      L     #Ziel;
      <=I;
      JC    chkl;
      CAC;
chkl: L     "DB_POS".LENG;
      *I;
      L     "DB_POS".Offset;
      +I;
      SLD   3;
      LAR1;
      OPN   "DB_POS";
      L     DBD [AR1, P#22.0];  //BadPos in Inkrementen
      L     #ZielInc;
      >D;
      R     #temp_erlaubt;
      JC    ende;
      JU    retl;


NETWORK
TITLE = nach rechts (zum höheren) suchen
//Es existiert rechts kein FW
sre:  A     #high_FW;
      JC    QT;

//-----------------------------------------
//größtes Ziel PosInc laden
      L     #temp_Gr_Z;
      L     "DB_POS".LENG;
      *I;
      L     "DB_POS".Offset;
      +I;
      SLD   3;
      LAR1;
      OPN   "DB_POS";
      L     DBD [AR1, P#22.0];  //BadPos in Inkrementen
      T     #PosmitteInc;
      AN    #Ablassen;
      JC    nab2;
      L     DBD [AR1, P#64.0];  //"DB_POS".POS[0].SonderPos_Offset
      +D;
nab2: T     #ZielInc;
//-----------------------------------------

//-----------------------------------------
//Start-FW laden
      L     #FW_Nr;
      T     #FW_count;
      L     10;
      +I;
      T     #FW_DB;

      OPN   DB [#FW_DB];
      L     #ZielInc;
      L     %DBD212;  //"DI_FW_1".PAR.Fahrt.Bereich_Pos
      +D;
      T     #ZielInc;

      OPN   DB [#FW_DB];
      L     %DBB186;  //"DI_FW_1".PAR.Reihe
      T     #Row;
      L     0;
      ==I;
      =     #nRowChk;

      OPN   DB [#FW_DB];
      L     %DBB2;  //"DI_FW_1".ZST.POSITION
      T     #IstPos;
      L     %DBD4;  //"DI_FW_1".ZST.PosInc
      T     #IstInc;
      L     %DBD212;  //"DI_FW_1".PAR.Fahrt.Bereich_Pos
      T     #PosBereich;
//-----------------------------------------

//-----------------------------------------
//Bewegt sich der zu prüfende TW
//immer in Richtung kleinere Position
      L     #PosmitteInc;
      L     #PosBereich;
      -D;
      L     #IstInc;
      <=D;
      A(;
      L     #IstPos;
      L     #temp_Gr_Z;
      >=I;
      );
      AN(;
      L     #temp_kl_Z;
      L     #temp_Gr_Z;
      ==I;
      );
      AN    #vor;
      A     #chk_on;
      JC    QT;
//-----------------------------------------

//-----------------------------------------
//Nachbar-FW prüfen
retr: L     #FW_count;
      L     10;
      +I;
      T     #FW_DB;
      OPN   DB [#FW_DB];
      L     #ZielInc;
      L     %DBD198;  //"DI_FW_2".PAR.Fahrt.Abstand_vor
      +D;
      T     #ZielInc;

      L     #FW_count;
      +     1;
      T     #FW_count;
      L     "DB_ANLAGE".config.ANZ_FW;
      >I;
      JC    QT;

      L     #FW_count;
      L     10;
      +I;
      T     #FW_DB;
      OPN   DB [#FW_DB];
//-----------------------------------------

//-----------------------------------------
//Reihe prüfen
      A     #nRowChk;
      JC    nRr;
      L     0;
      L     %DBB186;  //"DI_FW_1".PAR.Reihe
      ==I;
      S     #nRowChk;
      JC    nRr;
      L     #Row;  //Ende der Reihe
      <>I;
      JC    QT;
//-----------------------------------------

//-----------------------------------------
//Zielinkrement korrigieren
nRr:  L     #ZielInc;
      L     %DBD212;  //"DI_FW_1".PAR.Fahrt.Bereich_Pos
      +D;
      T     #ZielInc;
//-----------------------------------------

//-----------------------------------------
//Quelle/Ziel prüfen
      L     %DBB32;
      T     #Quelle;
      L     %DBB33;
      T     #Ziel;
      L     %DBB351;  //"DI_FW_1".TMP.ZielPos
      T     #aktZiel;
      A     %DBX0.6;  //"DI_FW_1".ZST.VORWAERTS_AKT
      =     #vor_akt;

      L     #Ziel;
      L     0;
      ==I;
      A(;
      L     #Quelle;
      <>I;
      );
      JCN   okr;
      T     #Ziel;
      L     0;
      T     #Quelle;

//-----------------------------------------

//-----------------------------------------
//FW muss geschoben werden
okr:  L     #Quelle;
      L     #Ziel;
      +I;
      L     0;
      ==I;
      O(;
      L     #aktZiel;
      L     #Ziel;
      ==I;
      A(;
      L     %DBB2;  //"DI_FW_1".ZST.POSITION
      ==I;
      A     %DBX53.2;  //"DI_FW_1".IN.Pos_ok
      AN    %DBX0.7;  //"DI_FW_1".ZST.RUECKWAERTS_AKT
      );
      );
      =     #TW_in_Quelle;
      JC    sLi;

//neu Test Nachfahren
      L     #Quelle;  //Lerfahrt
      L     0;
      ==I;
      =     #Q_null;

      L     #Quelle;
      L     #Ziel;
      ==I;
      AN    #TW_in_Quelle;
      JC    sLi;

      L     #aktZiel;
      L     #Ziel;
      ==I;
      A(;
      L     #Quelle;
      >=I;
      AN    #Q_null;
      O(;
      A     #Q_null;
      A     #vor_akt;
      );
      );
      JC    sLi;
      JU    nSLi;

sLi:  L     #temp_Gr_Z;
rpor: T     #Quelle;
      L     "DB_ANLAGE".config.ANZ_Pos;
      >I;
      R     #temp_erlaubt;
      JC    ende;

      L     #Quelle;
      L     "DB_POS".LENG;
      *I;
      L     "DB_POS".Offset;
      +I;
      SLD   3;
      LAR1;
      OPN   "DB_POS";
//Reihe zu ende?
      A     #nRowChk;
      JC    spor;
      L     DBB [AR1, P#4.0];  //"DB_POS".POS[0].Reihe
      L     #Row;
      <>I;
      R     #temp_erlaubt;
      JC    ende;

//mögliche Schiebepos?
spor: L     #ZielInc;
      L     DBD [AR1, P#22.0];  //BadPos in Inkrementen
      >D;
      JC    nxQr;
      T     #ZielInc;
      JU    retr;

nxQr: L     #Quelle;
      +     1;
      JU    rpor;
//-----------------------------------------

//-----------------------------------------
nSLi: L     0;
      L     #Ziel;
      ==I;
      JC    tstr;  //Leerfahrt- oder Schiebebefehl
      L     #aktZiel;
      ==I;
      JC    chkr;  //Quelle bereits bedient
tstr: L     #Quelle;
      L     #Ziel;
      >=I;
      JC    chkr;
      CAC;
chkr: L     "DB_POS".LENG;
      *I;
      L     "DB_POS".Offset;
      +I;
      SLD   3;
      LAR1;
      OPN   "DB_POS";
      L     DBD [AR1, P#22.0];  //BadPos in Inkrementen
      L     #ZielInc;
      <D;
      R     #temp_erlaubt;
      JC    ende;
      JU    retr;


NETWORK
TITLE = Test QT
//QT reserviert Bad für Transport
//daher Fahrbereich auf reserviertes Bad prüfen
//Sperre wird bei ankommenden Befehl gesetzt
//und wieder zurückgenommen, wenn sich der QT in bewegung setzt.
//Dann ist die Überfahrt durch FWs gesperrt.

QT:   AN    #QT_Check;
      JC    out;  //BEB

      A     #temp_erlaubt;
      =     #temp_erlaubt;

      L     #FW_Nr;
      L     10;
      +I;
      T     #FW_DB;

//FW Position laden
      OPN   DB [#FW_DB];
      L     %DBB2;  //"DBI_FW_1".ZST.POSITION
      T     #Quelle;

//Fahrbereich aufspannen
      L     #temp_Gr_Z;
      L     #Quelle;
      >=I;
      JC    klZ;
      T     #temp_Gr_Z;
klZ:  L     #temp_kl_Z;
      L     #Quelle;
      <=I;
      JC    test;
      T     #temp_kl_Z;

//Fahrbereich von größter Position bis kleinster prüfen
test: L     #temp_Gr_Z;
      L     "DB_POS".LENG;
      *I;
      L     "DB_POS".Offset;
      +I;
      SLD   3;
      LAR1;

      OPN   "DB_POS";
      L     DBB [AR1, P#0.0];  //PosTp QT?
      L     10;
      ==I;
      A     DBX [AR1, P#7.7];  //QT Reservierung
      R     #temp_erlaubt;

      L     #temp_Gr_Z;
      L     #temp_kl_Z;
      <=I;
      JC    ende;

      L     #temp_Gr_Z;
      L     1;
      -I;
      T     #temp_Gr_Z;
      JU    test;


NETWORK
TITLE = Adressregister zurückladen
ende: L     #Save_AR1;
      LAR1;
      L     #Save_AR2;
      LAR2;

NETWORK
TITLE = Out beschreiben
out:  A     #temp_erlaubt;
      =     #erlaubt;

END_FUNCTION

FUNCTION_BLOCK "FB_QF"   // FB31, LAD
TITLE = Querförderer
{ S7_Optimized_Access := 'TRUE' }
// stored: AutoNumber false, MemoryReserve 100, SetENOAutomatically true
   VAR RETAIN
      In { ExternalAccessible := 'False'; ExternalVisible := 'False'; ExternalWritable := 'False'} : Struct
         NotHalt : Bool;
         Auto : Bool;
         Hand : Bool;
         Tipp : Bool;
         T_WR02_zu_UE : Bool;
         T_WR02_zu_BE : Bool;
         T_WR03_zu_UE : Bool;
         T_WR03_zu_BE : Bool;
         S_WR02_lgsm_UE : Bool;
         S_WR02_lgsm_BE : Bool;
         S_WR03_lgsm_UE : Bool;
         S_WR03_lgsm_BE : Bool;
         S_WR02_UE : Bool;
         S_WR02_BE : Bool;
         S_WR03_UE : Bool;
         S_WR03_BE : Bool;
         Req_Ausfahrt_GO : Bool;
         Req_Aufgabe_GO : Bool;
         FU_betriebsbereit_WR02 : Bool;
         FU_betriebsbereit_WR03 : Bool;
         FU_Stoerung_WR02 : Bool;
         FU_Stoerung_WR03 : Bool;
         ErrQ : Bool;
         FU_speed_WR02 : Int;
         FU_speed_WR03 : Int;
      END_STRUCT;
      Param { ExternalAccessible := 'False'; ExternalVisible := 'False'; ExternalWritable := 'False'} : Struct
         "TO" : Time := T#48s;
      END_STRUCT;
      Zst { ExternalAccessible := 'False'; ExternalVisible := 'False'; ExternalWritable := 'False'} : Struct
         Fehler : Bool;
         Req_WR02_In : Bool;
         Req_WR03_In : Bool;
         Req_WR02_Out : Bool;
         Req_WR03_Out : Bool;
         Tor_sicher : Bool;
         TW_sicher : Bool;
      END_STRUCT;
      Out { ExternalAccessible := 'False'; ExternalVisible := 'False'; ExternalWritable := 'False'} : Struct
         WR02_einfahren : Bool;   // zur ÜbergabeStation
         WR02_ausfahren : Bool;   // zum Be-/Entladen
         WR03_einfahren : Bool;   // zur ÜbergabeStation
         WR03_ausfahren : Bool;   // zum Be-/Entladen
         Soll_speed_WR02 : Int;
         Soll_speed_WR03 : Int;
      END_STRUCT;
      Mld { ExternalAccessible := 'False'; ExternalVisible := 'False'; ExternalWritable := 'False'} : Struct
         TO_WR02 : Bool;
         TO_WR03 : Bool;
         St_FU_WR02 : Bool;
         St_FU_WR03 : Bool;
         FU_nichtbereit_WR02 : Bool;
         FU_nichtbereit_WR03 : Bool;
         n_Auto : Bool;
         SF_WR02 : Bool;
         SF_WR03 : Bool;
      END_STRUCT;
   END_VAR
   VAR
      IEC_Timer { ExternalAccessible := 'False'; ExternalVisible := 'False'; ExternalWritable := 'False'} : Struct
         TO_WR02 { S7_SetPoint := 'True'} : TON_TIME;
         TO_WR03 { S7_SetPoint := 'True'} : TON_TIME;
      END_STRUCT;
   END_VAR
   VAR_TEMP
      TO_WR02 : Bool;
      TO_WR03 : Bool;
   END_VAR
   VAR CONSTANT
      Speed_Tipp : Int := 25;   // %
      Speed_Hand : Int := 70;   // %
      Speed_Auto : Int := 70;   // % == 35 Hz = 150 mm/s
   END_VAR
BEGIN

REGION Network 1 (SCL): Input
   // Panelbedienung und Sensoren --> Input()
   // Not-Halt
   #In.NotHalt := NOT "DB_PNOZ_IN_Out".In.NH_Frg_TW_QF;
   // Rolltor
   #Zst.Tor_sicher := "Tor".In.S_auf AND NOT "Tor".Out.zu;
   // Transportwagen 
   #Zst.TW_sicher := "DI_FW_1".ZST.PosInc < ("DB_POS".POS[25].IncPos - "DB_POS".POS[25].IncAbstand_rck);

   // Anforderung Automatikbetrieb
   IF #In.Auto THEN
       "FC_Anf_BE"(Req_GO_Ausfahrt := #In.Req_Ausfahrt_GO,
                   Req_GO_Aufgabe := #In.Req_Aufgabe_GO,
                   Req_WR02_IN := #Zst.Req_WR02_In,
                   Req_WR02_OUT := #Zst.Req_WR02_Out,
                   Req_WR03_IN := #Zst.Req_WR03_In,
                   Req_WR03_OUT := #Zst.Req_WR03_Out);
   ELSE
       #Zst.Req_WR02_In := FALSE;
       #Zst.Req_WR02_Out := FALSE;
       #Zst.Req_WR03_In := FALSE;
       #Zst.Req_WR03_Out := FALSE;
   END_IF;
END_REGION

REGION Network 2 (SCL): Sammelstörung
   IF #In.ErrQ THEN
       #Zst.Fehler := FALSE;
   END_IF;

   IF #In.NotHalt OR #Mld.FU_nichtbereit_WR02 OR #Mld.FU_nichtbereit_WR03 OR #Mld.SF_WR02
       OR #Mld.SF_WR03 OR #Mld.St_FU_WR02 OR #Mld.St_FU_WR03 OR #Mld.TO_WR02 OR #Mld.TO_WR03  THEN
       #Zst.Fehler := TRUE;
   END_IF;
END_REGION

REGION Network 3 (SCL): Ansteuerung
   IF NOT #Zst.Fehler AND #Zst.Tor_sicher AND #Zst.TW_sicher THEN
       IF #In.Auto THEN // Automatikbetrieb
           // WR02
           #Out.WR02_einfahren := #Zst.Req_WR02_In;
           #Out.WR02_ausfahren := #Zst.Req_WR02_Out;
           // WR03
           #Out.WR03_einfahren := #Zst.Req_WR03_In;
           #Out.WR03_ausfahren := #Zst.Req_WR03_Out;

       ELSIF #In.Hand THEN // Handbetrieb

           // WR02
           IF #In.T_WR02_zu_UE AND NOT #In.T_WR02_zu_BE THEN
               #Out.WR02_einfahren := TRUE;
               #Out.WR02_ausfahren := FALSE;
           END_IF;
           IF #In.T_WR02_zu_BE AND NOT #In.T_WR02_zu_UE THEN
               #Out.WR02_ausfahren := TRUE;
               #Out.WR02_einfahren := FALSE;
           END_IF;
           // WR03
           IF #In.T_WR03_zu_UE AND NOT #In.T_WR03_zu_BE THEN
               #Out.WR03_einfahren := TRUE;
               #Out.WR03_ausfahren := FALSE;
           END_IF;
           IF #In.T_WR03_zu_BE AND NOT #In.T_WR03_zu_UE THEN
               #Out.WR03_ausfahren := TRUE;
               #Out.WR03_einfahren := FALSE;
           END_IF;
       ELSIF #In.Tipp THEN  // Tippbetrieb
           // WR02
           #Out.WR02_einfahren := #In.T_WR02_zu_UE AND NOT #In.T_WR02_zu_BE;
           #Out.WR02_ausfahren := #In.T_WR02_zu_BE AND NOT #In.T_WR02_zu_UE;

           // WR03
           #Out.WR03_einfahren := #In.T_WR03_zu_UE AND NOT #In.T_WR03_zu_BE;
           #Out.WR03_ausfahren := #In.T_WR03_zu_BE AND NOT #In.T_WR03_zu_UE;
       ELSE
           #Out.WR02_einfahren := FALSE;
           #Out.WR02_ausfahren := FALSE;
           #Out.WR03_einfahren := FALSE;
           #Out.WR03_ausfahren := FALSE;

       END_IF;

   ELSE // Not-Halt
       #Out.WR02_einfahren := FALSE;
       #Out.WR02_ausfahren := FALSE;
       #Out.WR03_einfahren := FALSE;
       #Out.WR03_ausfahren := FALSE;

   END_IF;

   // Endlagen erreicht
   IF #In.S_WR02_UE THEN
       #Out.WR02_einfahren := FALSE;
       #Zst.Req_WR02_In := FALSE;
   END_IF;
   IF #In.S_WR02_BE THEN
       #Out.WR02_ausfahren := FALSE;
       #Zst.Req_WR02_Out := FALSE;
   END_IF;
   IF #In.S_WR03_UE THEN
       #Out.WR03_einfahren := FALSE;
       #Zst.Req_WR03_In := FALSE;
   END_IF;
   IF #In.S_WR03_BE THEN
       #Out.WR03_ausfahren := FALSE;
       #Zst.Req_WR03_Out := FALSE;
   END_IF;

   // Geschwindigkeitsvorgabe WR02
   IF NOT #Out.WR02_einfahren AND NOT #Out.WR02_ausfahren THEN
       #Out.Soll_speed_WR02 := 0;
   ELSIF #In.Tipp THEN
       #Out.Soll_speed_WR02 := #Speed_Tipp;
   ELSIF #In.Hand THEN
       #Out.Soll_speed_WR02 := #Speed_Hand;
   ELSE
       #Out.Soll_speed_WR02 := #Speed_Auto;
   END_IF;
   // Positionierung
   IF (#Out.WR02_einfahren AND #In.S_WR02_lgsm_UE) OR (#Out.WR02_ausfahren AND #In.S_WR02_lgsm_BE)THEN
       #Out.Soll_speed_WR02 := #Speed_Tipp;
   END_IF;

   // Geschwindigkeitsvorgabe WR03
   IF NOT #Out.WR03_einfahren AND NOT #Out.WR03_ausfahren THEN
       #Out.Soll_speed_WR03 := 0;
   ELSIF #In.Tipp THEN
       #Out.Soll_speed_WR03 := #Speed_Tipp;
   ELSIF #In.Hand THEN
       #Out.Soll_speed_WR03 := #Speed_Hand;
   ELSE
       #Out.Soll_speed_WR03 := #Speed_Auto;
   END_IF;
   // Positionierung
   IF (#Out.WR03_einfahren AND #In.S_WR03_lgsm_UE) OR (#Out.WR03_ausfahren AND #In.S_WR03_lgsm_BE) THEN
       #Out.Soll_speed_WR03 := #Speed_Tipp;
   END_IF;
END_REGION

REGION Network 4 (SCL): Überwachung / Alarme
   // Störung FU WR02
   #Mld.St_FU_WR02 := #In.FU_Stoerung_WR02 AND NOT #In.NotHalt;
   // Störung FU WR03
   #Mld.St_FU_WR03 := #In.FU_Stoerung_WR03 AND NOT #In.NotHalt;
   // 24V-Betrieb
   #Mld.FU_nichtbereit_WR02 := NOT #In.FU_betriebsbereit_WR02 AND NOT #In.NotHalt;
   #Mld.FU_nichtbereit_WR03 := NOT #In.FU_betriebsbereit_WR03 AND NOT #In.NotHalt;

   // nicht in Automatik
   #Mld.n_Auto := NOT #In.Auto AND "DB_ANLAGE".BA.Automat_ein;

   // Zeitüberschreitung WR02
   #IEC_Timer.TO_WR02(IN := (#Out.WR02_einfahren AND NOT #In.S_WR02_UE) OR (#Out.WR02_ausfahren AND NOT #In.S_WR02_BE),
                        PT := #Param.TO,
                        Q => #TO_WR02);
     IF #TO_WR02 AND #In.Auto THEN
         #Mld.TO_WR02 := TRUE;
     ELSIF #In.ErrQ THEN
         #Mld.TO_WR02 := FALSE;
     END_IF;
   // Zeitüberschreitung WR03
     #IEC_Timer.TO_WR02(IN := (#Out.WR03_einfahren AND NOT #In.S_WR03_UE) OR (#Out.WR03_ausfahren AND NOT #In.S_WR03_BE),
                        PT := #Param.TO,
                        Q => #TO_WR03);
     IF #TO_WR03 AND #In.Auto THEN
         #Mld.TO_WR03 := TRUE;
     ELSIF #In.ErrQ THEN
         #Mld.TO_WR03 := FALSE;
     END_IF;
     //Sensorfehler
     #Mld.SF_WR02 := #In.S_WR02_UE AND #In.S_WR02_BE;
     #Mld.SF_WR03 := #In.S_WR03_UE AND #In.S_WR03_BE;
END_REGION
END_FUNCTION_BLOCK

FUNCTION "FC_Pos_Manager" : Void   // FC50, STL
TITLE = Positionsmanager
{ S7_Optimized_Access := 'FALSE' }
// Bearbeitung und Aktualisierung der Positionen
// in jedem Zyklus wird eine im DB1 definierte Anzahl von Positionen bearbeitet.
// stored: AutoNumber false
   VAR_TEMP
      count : Int;   // Zähler Pos pro Zyklus
      akt_Pos : USInt;   // aktuelle Position
      DummyPos : Bool;   // Position nicht behandeln
   END_VAR
BEGIN

NETWORK
TITLE = Umlauf Pos per Zyklus
// Umlaufzähler verwalten für Positionsbearbeitung
//----------------------------------
//Umlauf
//----------------------------------
      L     "DB_ANLAGE".config.ANZ_POS_per_Cyc;
schl: T     #count;

      L     "DB_POS".akt_POS;
      L     1;
      <I;
      JC    nok;
      L     "DB_POS".akt_POS;
      L     "DB_ANLAGE".config.ANZ_Pos;
      <=I;
      JC    go;

nok:  L     1;
      T     "DB_POS".akt_POS;

go:   L     "DB_POS".akt_POS;
      T     #akt_Pos;
//---------------------------------
//laden der Positionsdaten
//---------------------------------
      CALL  "FC_POS_TO_WORK"
      ( Akt_Pos  := #akt_Pos,
        not_load := #DummyPos
      );

//----------------------------------
//Position geladen --> Behandlung
//----------------------------------
      A     #DummyPos;
      JC    nexP;


NETWORK
TITLE = Badbehandlung
// Bearbeitung der Positionen und Aktualisierung von PC-Daten

      CALL  "FC_Pos_Behandlung"
      ( Pos_Nr     := #akt_Pos,
        send_DBEvt := TRUE
      );


NETWORK
TITLE = Rückladen der Positionsdaten
// Daten werden aus dem Arbeitsbereich wieder ausgelagert
//----------------------------------
//zurück laden der Positionsdaten
//----------------------------------
      CALL  "FC_WORK_TO_POS"
      ( Akt_Pos := #akt_Pos
      );
//----------------------------------
//Zeiger auf nächste Position setzen
//----------------------------------
nexP: L     "DB_POS".akt_POS;
      L     1;
      +I;
      T     "DB_POS".akt_POS;
//----------------------------------
//Zählschleifenrücksprung
//----------------------------------
      L     #count;
      LOOP  schl;
      BE;
END_FUNCTION

FUNCTION "FC_Zaehler" : Void   // FC80, STL
TITLE = FC_LADUZA
{ S7_Optimized_Access := 'FALSE' }
AUTHOR : KHE
NAME : FC_LADUN
// Dosierzaehler
// stored: AutoNumber false
   VAR_TEMP
      DPOIN1 : DWord;   // Datenpointer 1
      DPOIN2 : DWord;   // Datenpointer 2
      Z_Summe : DWord;   // Zwischensumme
      AR1 : DWord;   // Puffer AR1
      Param : DWord;
      Korfa : Real;   // Korrekturfaktor
      Intervall : DInt;
      B_BAD : Byte;
      GR_2 : Byte;
      Am_Zaehler : Bool;   // AmpereMinuten-Ladungszählung
      dm2_Zaehler : Bool;   // Oberflächenzählung
      WT_Zaehler : Bool;   // Warenträgerzählung
      Ext_Zaehler : Bool;   // Externe Zählung
      Sond_Zaehl : Bool;   // Sonderzähler EJOT2
      Ext_Ah_Zae : Bool;   // externer Ah-Zähler
      aktual : Bool;   // Wert aktualisieren
      belegt : Bool;
      GR2_run : Bool;
      Evt : Bool;
      ohne_Pos : Bool;
      leerWt : Bool;
      Belegt_GO : Bool;
   END_VAR
BEGIN

NETWORK
TITLE = Start
// Initialisierung und Taktung

      A     "Imp_1Hz";
      JCN   takt;

      L     "DB_Zaehler".I_Time;  //Integrationszeit
      INC   1;
      T     "DB_Zaehler".I_Time;  //Integrationszeit

takt: L     "DB_Zaehler".I_Time;
      L     0;
      ==I;
      JC    exit;
      L     "DB_Zaehler".Anz_Beck;  //Becken-Anz.
      >=I;
      JC    exit;
      L     "DB_Zaehler".Beck_Nr;  //Becken-Pointer
      INC   1;
      >=I;
      JC    bec1;
      L     "DB_Zaehler".I_Time;
      DEC   1;
      T     "DB_Zaehler".I_Time;
      L     0;
      T     "DB_Zaehler".Beck_Nr;

//Events intern ----------------------------
//-- Ta/Wo-Za ----------
      L     "DB_Zaehler".MZ_T;
      L     "Uhrzeit".aktDatum.DAY;  //akt.Tag [DT]
      ==I;
      JC    tzx;
      T     "DB_Zaehler".MZ_T;
      L     "Uhrzeit".aktDatum.WEEKDAY;  //akt.Tag der Woche [DT]
      L     1;  //Sonntag
      <>I;
      JC    wzx;
      S     "DB_Zaehler".Wo_neu;
wzx:  CLR;
tzx:  R     "DB_Zaehler".Wo_neu;
      NOT;
      =     "DB_Zaehler".Tag_neu;

//-- Mo-Za ----------
      L     "DB_Zaehler".MZ_M;
      L     "Uhrzeit".aktDatum.MONTH;  //akt.Monat [DT]
      ==I;
      JC    mzx;
      T     "DB_Zaehler".MZ_M;
      CLR;
mzx:  NOT;
      =     "DB_Zaehler".Mo_neu;
      JU    exit;

//------------------------------------
bec1: T     "DB_Zaehler".Beck_Nr;
      +     -1;
      L     "DB_Zaehler".leng_Pos;
      *D;
      L     "DB_Zaehler".Offset;
      +D;
      SLD   3;  //Korr. f. Pointer
      LAR1;
      OPN   "DB_Zaehler";
      T     #DPOIN1;

      A     DBX [AR1, P#27.7];  //Anf_Stp
      R     DBX [AR1, P#27.7];  //Anf_Stp
      =     DBX [AR1, P#27.1];  //Stop

//-- Init ------------------------
      L     0.0;
      T     #Z_Summe;
      L     0;
      T     #B_BAD;
      CLR;
      =     #Evt;
      =     #ohne_Pos;

      L     DBB [#DPOIN1];  //Typ
      L     1;
      ==I;
      =     #Am_Zaehler;
      POP;
      L     4;
      ==I;
      =     #dm2_Zaehler;
      POP;
      L     5;
      ==I;
      =     #WT_Zaehler;
      POP;
      L     6;
      ==I;
      =     #Ext_Zaehler;
      S     #ohne_Pos;
      POP;
      L     7;
      ==I;
      =     #Sond_Zaehl;
      S     #ohne_Pos;
      POP;
      L     8;
      ==I;
      =     #Ext_Ah_Zae;
      S     #ohne_Pos;


NETWORK
TITLE = MeZa
// Mengenzähler, allgemein
      AN    #Sond_Zaehl;
      JC    extZ;

      OPN   "DB_Zaehler";
      L     DBD [AR1, P#34.0];  //"DB_LZ".Becken[1].ext_Val
      T     #Z_Summe;
      L     1.0;
      T     #Korfa;
      L     0.0;
      T     DBD [AR1, P#34.0];  //"DB_LZ".Becken[1].ext_Val
      JU    ext;

extZ: AN    #Ext_Zaehler;
      JC    loop;
//ext.Zähler über Event (FC6) --------------------
      L     0;
      L     "DB_Zaehler".Beck_ext;
      ==I;
      JC    exit;
      L     "DB_Zaehler".Beck_Nr;
      <>I;
      JC    exit;
      L     "DB_Zaehler".Wert_Ext;
      T     #Z_Summe;
      L     0;
      T     "DB_Zaehler".Beck_ext;
      JU    korr;

//----------- Dosierz. Werte aus Bädern aufaddieren-----
loop: OPN   "DB_Zaehler";  //Arbeits-DB
      L     DBB [AR1, P#1.0];  //Anz. Pos. je Becken
      L     #B_BAD;
      <=I;
      JC    korr;
      INC   1;
      T     #B_BAD;
      L     #DPOIN1;
      L     2;  //Offset Pos.-Nr
      SLD   3;
      +D;
      T     #DPOIN1;
      L     0;
      L     DBW [#DPOIN1];
      >=I;
      JC    loop;

//---- Badpointer -------------
      L     "DB_POS".LENG;
      *D;
      L     "DB_POS".Offset;
      +D;
      SLD   3;
      LAR2;
      OPN   "DB_POS";
      A     DBX [AR2, P#96.0];  //belegt
      =     #belegt;
      A     DBX [AR2, P#38.1];  //leer WT
      =     #leerWt;
      A     DBX [AR2, P#8.5];  //"DB_POS".POS[x].Belegt_GO
      =     #Belegt_GO;
      TAR1;
      L     "DB_Zaehler".leng_Pos;
      +     -2;  //letzten 2Byte in LZ
      SLD   3;
      +D;  //Offset AM-bel
      L     #B_BAD;
      DEC   1;
      +D;
      T     #DPOIN2;
      OPN   "DB_Zaehler";
      AN    #belegt;
      A     DBX [#DPOIN2];
      =     #aktual;
      S     #Evt;
      A     #belegt;
      =     DBX [#DPOIN2];

      A     #dm2_Zaehler;
      O     #WT_Zaehler;
      JC    OF;

OF:   AN    #aktual;
      JC    loop;
      A     #WT_Zaehler;
      A     #leerWt;
      JC    loop;
      L     1.0;  //1x WT
      A     #WT_Zaehler;
      AN    #Belegt_GO;
      JC    add;
      L     2.0;  //2x WT - GO doppelt zählen
      A     #WT_Zaehler;
      A     #Belegt_GO;
      JC    add;
      OPN   "DB_POS";
      L     DBD [AR2, P#52.0];  //Oberfläche
add:  L     #Z_Summe;
      +R;
Off:  T     #Z_Summe;

      A     #dm2_Zaehler;
      O     #WT_Zaehler;
      JC    loop;
      JU    loop;

//Korrektur-Rechnung ---------------------------
korr: L     1.0;  //Flächenfaktor
      A     #dm2_Zaehler;
      O     #WT_Zaehler;
      O     #Ext_Zaehler;
      JC    kor2;
      L     60.0;  //60 (sec->min)
      A     #Am_Zaehler;
      JC    kor2;
      L     3600.0;  //3600 (sec->h)
kor2: T     #Korfa;

ext:  OPN   "DB_Zaehler";
      L     #Z_Summe;
      L     DBD [AR1, P#22.0];  //Zwischen-Zähler
      +R;
      T     DBD [AR1, P#22.0];  //Zwischen-Zähler
      L     #Korfa;
      /R;  //Asec->Ah
      TRUNC;  //GP->DINT
      T     #Z_Summe;
      DTR;  //DINT->GP
      L     #Korfa;
      *R;
      L     DBD [AR1, P#22.0];  //Zwischen-Zähler
      CAC;
      -R;
      T     DBD [AR1, P#22.0];  //Zwischen-Zähler


NETWORK
TITLE = Zähler
// Zähler und ihre Auswertung
      L     "DB_Zaehler".Beck_Nr;
      L     1;
      -D;
      L     "DB_Panel_LZ".Length;
      *D;
      L     "DB_Panel_LZ".Offset;
      +D;
      SLD   3;  //Korr. f. Pointer
      LAR2;

      OPN   "DB_Zaehler";
      L     DBD [AR1, P#30.0];  //"DB_LZ".Becken[1].EventCount
      L     #Z_Summe;
      +D;
      T     DBD [AR1, P#30.0];  //"DB_LZ".Becken[1].EventCount

// Restzähler ---------------------------------------
      OPN   "DB_Zaehler";
      L     DBD [AR1, P#22.0];  //A-sec-Zähler
      RND;  //GP->DINT
      OPN   "DB_Panel_LZ";
      T     DBD [AR2, P#8.0];  //Rest_Zaehl

// Aktual. Dosi.Zaehler --------------------------------
      L     DBD [AR2, P#4.0];  //Dosi_Zaehl
      L     #Z_Summe;
      +D;
      T     DBD [AR2, P#4.0];  //Dosi_Zaehl

// Aktual. Lad.Zähler 1 -------------------------------
      L     DBD [AR2, P#12.0];  //Ladu_Zaehl_1
      L     #Z_Summe;
      +D;
      T     DBD [AR2, P#12.0];  //Ladu_Zaehl_1

// Aktual. Lad.Zähler 2 -------------------------------
      L     DBD [AR2, P#16.0];  //Ladu_Zaehl_2
      L     #Z_Summe;
      +D;
      T     DBD [AR2, P#16.0];  //Ladu_Zaehl_2

// Aktual. Lad.Zähler 3 -------------------------------
      L     DBD [AR2, P#20.0];  //Ladu_Zaehl_3
      L     #Z_Summe;
      +D;
      T     DBD [AR2, P#20.0];  //Ladu_Zaehl_3

// Aktual. Lad.Zähler 4 -------------------------------
      L     DBD [AR2, P#24.0];  //Ladu_Zaehl_4
      L     #Z_Summe;
      +D;
      T     DBD [AR2, P#24.0];  //Ladu_Zaehl_4

// Aktual. Lad.Zähler 5 -------------------------------
      L     DBD [AR2, P#28.0];  //Ladu_Zaehl_5
      L     #Z_Summe;
      +D;
      T     DBD [AR2, P#28.0];  //Ladu_Zaehl_5

// Aktual. Lad.Zähler 6 -------------------------------
      L     DBD [AR2, P#32.0];  //Ladu_Zaehl_4
      L     #Z_Summe;
      +D;
      T     DBD [AR2, P#32.0];  //Ladu_Zaehl_4

//======= Event-Erzeugung und -Behandlung =============
//----------- Dosierung --------------
      OPN   "DB_Zaehler";
      A     DBX [AR1, P#27.0];  //Event
      R     DBX [AR1, P#27.0];  //Event
      JC    doze;
      A     DBX [AR1, P#27.1];  //Stop
      JC    doze;
      OPN   "DB_Panel_LZ";
      L     0;
      L     DBD [AR2, P#0.0];  //Dosi_Int
      ==D;
      JC    doze;
      L     DBD [AR2, P#4.0];  //Dosi_Zaehl
      L     DBD [AR2, P#0.0];  //Dosi_Int
      <D;
      JC    doze;
      -D;
      T     DBD [AR2, P#4.0];  //Dosi_Zaehl
      SET;
      OPN   "DB_Zaehler";
      S     DBX [AR1, P#27.0];  //Event
      A     #ohne_Pos;
      S     #Evt;
doze: SET;
//---------- Tageszähler --------------
      AN    "DB_Zaehler".Tag_neu;
      JC    tze;

      OPN   "DB_Panel_LZ";
//evtl umladen hier !!
//!
      L     0;
      T     DBD [AR2, P#12.0];  //Ladu_Zaehl_1
tze:  SET;

//---------- Wochenzähler --------------
      AN    "DB_Zaehler".Wo_neu;
      JC    wze;

      OPN   "DB_Panel_LZ";
//evtl umladen hier !!
//!
      L     0;
      T     DBD [AR2, P#16.0];  //Ladu_Zaehl_2
wze:  SET;

//---------- Monatszähler --------------
      AN    "DB_Zaehler".Mo_neu;
      JC    mze;

      OPN   "DB_Panel_LZ";
//evtl umladen hier !!
//!
      L     0;
      T     DBD [AR2, P#20.0];  //Ladu_Zaehl_3
mze:  SET;


//set Event-----------------------------
// hier eintragen


//Datenerfassung DB88--------------------
      AN    #Evt;
      JC    exit;
      OPN   "DB_Zaehler";
      L     DBD [AR1, P#30.0];  //"DB_LZ".Becken[1].EventCount
      T     #Intervall;
      DTR;
      T     #Param;
      L     "DB_Zaehler".Beck_Nr;
      T     #B_BAD;

      OPN   "DB_Zaehler";
      L     0;
      T     DBD [AR1, P#30.0];  //"DB_LZ".Becken[1].EventCount

      L     0;
      L     "DB_Zaehler".Beck_Nr;
      >=I;
      JC    exit;
      DEC   1;
      L     4;
      *D;
      SLD   3;
      LAR1;
      OPN   "DB_Dosi_Overview";
      L     DBD [AR1, P#0.0];
      L     #Intervall;
      +D;
      T     DBD [AR1, P#0.0];
exit: BE;

END_FUNCTION

FUNCTION "FC_DoPu" : Void   // FC85, STL
TITLE = Dosierpumpensteuerung
{ S7_Optimized_Access := 'FALSE' }
// stored: AutoNumber false
   VAR_TEMP
      Pumpleistung : Real;
      Handzugabe : Real;
      Autozugabe : Real;
      Restdosierwert : Real;
      Doswert : Real;
      Kalibrierwert : Real;
      Kali_Count : DInt;
      Adr_PC_DB : DWord;
      Param : DWord;
      leng_Platz : Int;
      Adr_Basis : Int;
      Adr_Pumpe : Int;
      count : Int;
      T_Impuls : Int;
      T_Pause : Int;
      AnzI : Int;
      Anz_DP : Int;
      DP_Nr : Byte;
      BA : USInt;
      LZ_NR : Byte;
      ON : Bool;
      Hand : Bool;
      AUTO : Bool;
      Kalibrierung : Bool;
      DP_An : Bool;
      EvtA : Bool;
      EvtH : Bool;
      Add : Bool;
      Check : Bool;   // Kontrollpumpe aktiviert
      Stoerung : Bool;
      New_Err : Bool;
      Kali_Start : Bool;
      Kali_Stop : Bool;
   END_VAR
BEGIN

NETWORK
TITLE = Initialisierung und Schleifensteuerung
      SET;
      =     "DB_ANLAGE".IN.pH_LF_ok;

      L     0;
      L     "DB_ANLAGE".config.Anz_DP;
      ==I;
      BEC;
      L     0;
      L     "DB_DP".CheckPU;
      <I;
      =     #Check;
      JCN   Cok;
      L     "DB_ANLAGE".config.Anz_DP;
      <=I;
      JC    Cok;
      R     #Check;
      L     0;
      T     "DB_DP".CheckPU;

Cok:  L     "DB_DP".leng_Pos;
      T     #leng_Platz;
      L     "DB_DP".Offset;
      T     #Adr_Basis;

      A     "Imp_1Hz";
      S     "DB_DP".Sekunden_Takt;

      L     0;
      L     "DB_DP".DP_Nr;
      <I;
      A(;
      L     "DB_DP".Anz_DP;
      <=I;
      );
      JC    go;
//-----------------------------------------
//Initialisierung nach einem Umlauf
//-----------------------------------------
      AN    "DB_DP".Sekunden_Takt;  //kein Umlaufstart
      JC    Out;  //zur Dosierung springen
      R     "DB_DP".Sekunden_Takt;

      L     "DB_ANLAGE".config.Anz_DP;
      T     "DB_DP".DP_Nr;

      L     "DB_DP".AM_Minute;
      L     "Uhrzeit".aktDatum.MINUTE;
      <>I;
      =     "DB_DP".Minuten_Takt;
      T     "DB_DP".AM_Minute;
      JCN   go;
      L     "DB_DP".MinCount;
      L     0;
      <=I;
      S     "DB_DP".HandeventTakt;
      L     15;
      JC    stEv;
      L     "DB_DP".MinCount;
      +     -1;
stEv: T     "DB_DP".MinCount;
//-----------------------------------------

go:   AN    #Check;
      L     "DB_DP".DP_Nr;
      JC    nC1;
      L     "DB_DP".CheckPU;
nC1:  L     #leng_Platz;
      *D;
      L     #Adr_Basis;
      +D;
      T     #Adr_Pumpe;

      CALL  "FC_Blk_Move"
      ( Quelle        := #Adr_Pumpe,
        Ziel          := #Adr_Basis,
        Laenge        := #leng_Platz,
        _InputBlockDB := "DB_DP"
      );
      JU    DZ;
//-----------------------------------------
//Ende der Bearbeitung einer Pumpe
//-----------------------------------------
EndP: CALL  "FC_Blk_Move"
      ( Quelle        := #Adr_Basis,
        Ziel          := #Adr_Pumpe,
        Laenge        := #leng_Platz,
        _InputBlockDB := "DB_DP"
      );

      A     #Check;
      JC    Out;

      L     "DB_DP".DP_Nr;
      +     -1;
      T     "DB_DP".DP_Nr;
      JU    Out;

NETWORK
TITLE = Dosierzählerdaten holen
DZ:   L     0;
      L     "DB_DP".DP[0].LaZa_Nr;  //externe Ansteuerung
      >=I;
      JC    EndP;
      L     "DB_ANLAGE".config.Anz_DZ;
      >I;
      JC    EndP;  //kein Dosierzähler zugeordnet
      CAC;
      +     -1;
      L     "DB_Zaehler".leng_Pos;
      *D;
      L     "DB_Zaehler".Offset;
      +D;
      SLD   3;  //Korr. f. Pointer
      LAR1;
      OPN   "DB_Zaehler";
      A     DBX [AR1, P#27.0];  //LaZa_Event
      =     "DB_DP".DP[0].DP_Start;
      JU    EndP;


NETWORK
TITLE = Ausgabe Dosierung
Out:  AN    "Imp_10Hz";  //1/10sec Takt
      BEC;

      A     #Check;
      L     "DB_DP".CheckPU;
      JC    retP;
      L     "DB_ANLAGE".config.Anz_DP;
retP: T     #count;
      L     #leng_Platz;
      *D;
      L     #Adr_Basis;
      +D;
      T     #Adr_Pumpe;

      L     #count;
      +     -1;
      L     "DB_Panel_DP".Length;
      *D;
      L     "DB_Panel_DP".Offset;
      +D;
      SLD   3;
      T     #Adr_PC_DB;

      CALL  "FC_Blk_Move"
      ( Quelle        := #Adr_Pumpe,
        Ziel          := #Adr_Basis,
        Laenge        := #leng_Platz,
        _InputBlockDB := "DB_DP"
      );
      JU    Pump;

nexP: CALL  "FC_Blk_Move"
      ( Quelle        := #Adr_Basis,
        Ziel          := #Adr_Pumpe,
        Laenge        := #leng_Platz,
        _InputBlockDB := "DB_DP"
      );

      A     #Check;
      JC    Chk1;

      L     #count;
      LOOP  retP;

Chk1: CLR;
      =     "DB_DP".Minuten_Takt;
      =     "DB_DP".HandeventTakt;
      BE;

NETWORK
TITLE = Dosierung melden
//-------------------------------------------
//Daten aus PC-DB holen
//-------------------------------------------
Pump: L     #Adr_PC_DB;
      LAR1;
      OPN   "DB_Panel_DP";
      A     DBX [AR1, P#6.0];  //"DB_PC_DP".DoPu[1].Ein
      =     #ON;
      A     DBX [AR1, P#6.1];  //"DB_PC_DP".DoPu[1].Auto
      =     #AUTO;
      A     DBX [AR1, P#6.2];  //"DB_PC_DP".DoPu[1].Kalibrierung
      =     #Kalibrierung;
      A     DBX [AR1, P#6.5];  //"DB_PC_DP".DoPu[1].Hand
      =     #Hand;
      A     DBX [AR1, P#6.6];  //"DB_PC_DP".DoPu[1].ON
      =     #DP_An;
      A     DBX [AR1, P#7.0];  //"DB_PC_DP".DoPu[1].Kali_Start
      =     #Kali_Start;
      A     DBX [AR1, P#7.1];  //"DB_PC_DP".DoPu[1].Kali_Stop
      =     #Kali_Stop;

      L     DBW [AR1, P#0.0];  //"DB_PC_DP".DoPu[1].Impulsdauer
      T     #T_Impuls;
      L     DBW [AR1, P#2.0];  //"DB_PC_DP".DoPu[1].Impulspause
      T     #T_Pause;
      L     DBD [AR1, P#8.0];  //"DB_PC_DP".DoPu[1].Pumpleistung
      T     #Pumpleistung;
      L     DBD [AR1, P#16.0];  //"DB_PC_DP".DoPu[1].Zugabe_Auto
      T     #Autozugabe;
      L     DBD [AR1, P#20.0];  //"DB_PC_DP".DoPu[1].RestDosierWert
      T     #Restdosierwert;
      L     DBD [AR1, P#24.0];  //"DB_PC_DP".DoPu[1].Kalibrierwert
      T     #Kalibrierwert;
      L     DBD [AR1, P#36.0];  //"DB_PC_DP".DoPu[1].Kali_Count
      T     #Kali_Count;

      L     DBD [AR1, P#12.0];  //"DB_PC_DP".DoPu[1].Handzugabe
//      L     "DB_DP".DP[0].DosMenge_Hand
//      -R
      T     #Handzugabe;

      L     "DB_DP".DP[0].ZeitBasis;
      L     1;  //Minute
      ==I;
      L     60.0;
      JC    Korr;
      L     "DB_DP".DP[0].ZeitBasis;
      L     2;
      ==I;
      L     3600.0;
      JC    Korr;
      JU    okTB;

Korr: L     #Pumpleistung;
      CAC;
      /R;
      T     #Pumpleistung;

okTB: A     #ON;
      O     #AUTO;
      O     #Hand;
      O     #Kalibrierung;
      A     "DB_DP".DP[0].DP_Strg;
      =     #Stoerung;

      A     "DB_DP".DP[0].DP_OFF;
      R     #DP_An;

//-------------------------------------------
//Kalibrierung
//-------------------------------------------
      A     #Kalibrierung;
      JC    Kal;
      L     0;
      T     #Kali_Count;
      JU    PuHA;

Kal:  L     "DB_DP".DP[0].Typ;
      JL    Lst;
      JU    KMPZ;  //0 Menge pro Zeit
      JU    KMPI;  //1 Menge pro Impuls
      JU    Lst;  //2
      JU    Lst;  //3
      JU    Lst;  //4
      JU    Lst;  //5
      JU    KMPM;  //6 Menge pro Minute
Lst:  L     0.0;
      T     #Doswert;
      SET;
      R     #Add;
      JU    KRun;

KMPZ: A     #Kali_Stop;
      R     #Kali_Stop;
      L     0;
      JC    SKC1;
      AN    #Kali_Start;
      JC    KSTR;
      R     #Kali_Start;
      L     #Kalibrierwert;
      L     10.0;
      *R;
      TRUNC;
      JU    SKC1;

KSTR: L     #Kali_Count;
      +     DINT#-1;
SKC1: T     #Kali_Count;
      JU    KRun;

KMPM: L     2;
      T     #T_Pause;

KMPI: A     #Kali_Stop;
      R     #Kali_Stop;
      L     0;
      JC    SKC2;
      AN    #Kali_Start;
      JC    KMSR;
      R     #Kali_Start;
      L     #Kalibrierwert;
      TRUNC;
      JU    SKC2;

KMSR: A     "DB_DP".DP[0].Dosi_akt;
      FN    "DB_DP".DP[0].AM_Dosi;
      JCN   KMZ1;
      L     #Kali_Count;
      +     DINT#-1;
SKC2: T     #Kali_Count;
KMZ1: JU    KRun;

KRun: L     #Kali_Count;
      L     0;
      <D;
      JC    SKC2;
      >D;
      AN    "DB_DP".DP[0].DP_OFF;
      =     #DP_An;
      JU    nEvt;

//-------------------------------------------
//Handevent bei Typ 2
//-------------------------------------------
PuHA: A     "DB_DP".HandeventTakt;
      S     "DB_DP".DP[0].Meldung;

//-------------------------------------------
//Automatikintervall zählen
//-------------------------------------------
      AN    "DB_DP".DP[0].DP_Start;
      JC    noIV;
      R     "DB_DP".DP[0].DP_Start;

      L     #Restdosierwert;
      L     #Autozugabe;
      +R;
      T     #Restdosierwert;

      L     "DB_DP".DP[0].Typ;
      L     2;
      ==I;
      S     "DB_DP".DP[0].Meldung;

noIV: NOP   0;
//-------------------------------------------
//Doswert für 100ms bzw. Impuls berechnen
//-------------------------------------------
      L     "DB_DP".DP[0].Typ;
      JL    list;
      JU    MPZ;  //0 Menge pro Zeit
      JU    MPI;  //1 Menge pro Impuls
      JU    MPH;  //2 Handzugabe ohne Pumpe
      JU    MxP;  //3 externer Impuls
      JU    list;  //4
      JU    H2O;  //5 Wassermengenzähler
list: L     0.0;
      T     #Doswert;
      SET;
      R     #Add;
      JU    DosA;

MPZ:  L     #Pumpleistung;
      L     10.0;
      /R;
      T     #Doswert;
      A     #DP_An;
      =     #Add;
      JU    DosA;

MPI:  A     "DB_DP".DP[0].Dosi_akt;
      FN    "DB_DP".DP[0].AM_Dosi;
      =     #Add;
      L     #Pumpleistung;
      T     #Doswert;
      JU    DosA;

MxP:  A     "DB_DP".DP[0].DP_Imp;
      FP    "DB_DP".DP[0].AM_Dosi;
      =     #Add;
      L     #Pumpleistung;
      T     #Doswert;
      JU    DosA;

MPH:  A     #Hand;
      =     #Add;
      L     0.0;
      JCN   noH;
      R     "DB_DP".DP[0].Meldung;
      L     #Handzugabe;
noH:  T     #Doswert;
      JU    DosA;

H2O:  L     #Restdosierwert;
      T     #Doswert;
      SET;
      =     #Add;
      JU    list;

//-------------------------------------------
//Dosmenge aufaddieren
//-------------------------------------------
DosA: AN    #Add;
      JC    nDos;

      AN    #Hand;
      JC    DAut;
      L     #Handzugabe;
      L     #Doswert;
      -R;
      T     #Handzugabe;

      L     "DB_DP".DP[0].Typ;  //bei man. Dosierzugabe
      L     2;  //wird auch der Restdosierwert reduziert
      ==I;
      JC    DAut;
      JU    DosC;

DAut: L     #Restdosierwert;
      L     #Doswert;
      -R;
      T     #Restdosierwert;
      L     0.0;
      >=R;
      JC    DosC;
      T     #Restdosierwert;

//Mengenzählung für PVS
DosC: A     #Hand;
      JC    DosH;
      L     "DB_DP".DP[0].DosMenge_Auto;
      L     #Doswert;
      +R;
      T     "DB_DP".DP[0].DosMenge_Auto;
      JU    DB88;

DosH: L     "DB_DP".DP[0].DosMenge_Hand;
      L     #Doswert;
      +R;
      T     "DB_DP".DP[0].DosMenge_Hand;

//Datenerfassung DB88----------------------------
//Offset Ladungszähler
DB88: L     "DB_Zaehler".Anz_Beck;
      L     4;
      *D;
      SLD   3;
      LAR1;

//Adresse Pumpe
      L     #count;
      DEC   1;
      L     8;
      *D;
      SLD   3;
      +AR1;

//je nach Betriebsart Zelle aufaddieren
      A     #Hand;
      JC    Add;
      +AR1  P#4.0;
Add:  OPN   "DB_Dosi_Overview";
      L     DBD [AR1, P#0.0];
      L     #Doswert;
      +R;
      T     DBD [AR1, P#0.0];

nDos: NOP   0;
//-------------------------------------------
//Betriebsart Dosierpumpe
//-------------------------------------------

//Handzugabe (immer erlaubt)
      AN    "DB_DP".DP[0].DP_Hand;
      R     #Hand;
      JC    BAA;
      L     #Handzugabe;
      L     #Doswert;
      <R;
      O     "DB_DP".DP[0].DP_Niv;
      O     "DB_DP".DP[0].DP_OFF;
      JC    delH;
      S     #Hand;
      S     #DP_An;
      JU    Evts;
delH: R     "DB_DP".DP[0].DP_Hand;
      R     #Hand;
      R     #DP_An;
      L     0.0;
      T     #Handzugabe;

//Pumpe AUS
BAA:  AN    #ON;
      AN    #AUTO;
      O     "DB_DP".DP[0].DP_Niv;
      R     #DP_An;
      JC    Evts;
//Pumpe EIN
      A     #ON;
      AN    #AUTO;
      AN    "DB_DP".DP[0].DP_OFF;
      S     #DP_An;
      JC    Evts;
//Automatik
      L     0.0;
      L     #Restdosierwert;
      <>R;
      A(;
      L     #Doswert;
      >=R;
      );
      AN    "DB_DP".DP[0].DP_OFF;
      =     #DP_An;

//-------------------------------------------
//Fehler-Event senden
//-------------------------------------------
      A     "DB_ANLAGE".IN.AMS_Restart;
      R     "DB_DP".DP[0].AM_Strg;

      A     #AUTO;
      O     #Hand;
      A     "DB_DP".DP[0].DP_Strg;
      =     #New_Err;
      A     "DB_DP".DP[0].DP_Strg;
      X     "DB_DP".DP[0].AM_Strg;
      JCN   ok;

      L     #count;
      T     #DP_Nr;
      L     "DB_DP".DP[0].LaZa_Nr;
      T     #LZ_NR;

      A     #New_Err;  //neuer Alarm --> Hupe an
      R     "DB_ANLAGE".config.M_Q_Hupe;

ok:   A     "DB_DP".DP[0].DP_Strg;
      =     "DB_DP".DP[0].AM_Strg;

//-------------------------------------------
//Event senden
//-------------------------------------------
Evts: AN    "DB_DP".Minuten_Takt;
      JC    HEv;
      L     "DB_DP".DP[0].Rest_EventTime;
      L     "DB_DP".DP[0].EventTime;
      >I;
      JC    HEv;
      L     "DB_DP".DP[0].Rest_EventTime;
      +     1;
      T     "DB_DP".DP[0].Rest_EventTime;

//Handevents
HEv:  L     0.0;
      L     "DB_DP".DP[0].DosMenge_Hand;
      <>R;
      AN    #Hand;
      =     #EvtH;

//Automatikevents
      L     "DB_DP".DP[0].Rest_EventTime;
      L     "DB_DP".DP[0].EventTime;
      >=R;
      AN    #DP_An;
      O     #Hand;
      =     #EvtA;

      L     0.0;
      L     "DB_DP".DP[0].DosMenge_Auto;
      ==R;
      R     #EvtA;

      A     #EvtA;
      JC    Auto;
      A     #EvtH;
      JC    Hand;
      JU    nEvt;

Auto: L     1;
      T     #BA;
      L     "DB_DP".DP[0].DosMenge_Auto;
      T     #Param;
      L     0.0;
      T     "DB_DP".DP[0].DosMenge_Auto;
      L     0;
      T     "DB_DP".DP[0].Rest_EventTime;
      JU    Evt;

Hand: L     2;
      T     #BA;
      L     "DB_DP".DP[0].DosMenge_Hand;
      T     #Param;
      L     0.0;
      T     "DB_DP".DP[0].DosMenge_Hand;

Evt:  L     #count;
      T     #DP_Nr;

nEvt: NOP   0;


NETWORK
TITLE = Pumpe ansteuern
      L     "DB_DP".DP[0].Typ;
      L     1;  //Impulspumpe
      ==I;
      JC    Imp;
      CAC;
      L     2;  //Handzugabe
      ==I;
      JC    HP;

      A     #DP_An;
      =     "DB_DP".DP[0].Dosi_akt;
      JU    Data;

Imp:  L     "DB_DP".DP[0].RestZeit;
      L     0;
      <=I;
      A     #DP_An;
      JC    OnOf;

      AN    #DP_An;
      A     "DB_DP".DP[0].Dosi_akt;
      JC    OnOf;

      L     "DB_DP".DP[0].RestZeit;
      L     0;
      <=I;
      JC    Data;

      L     "DB_DP".DP[0].RestZeit;
      +     -1;
      T     "DB_DP".DP[0].RestZeit;
      JU    Data;

OnOf: AN    "DB_DP".DP[0].Dosi_akt;
      =     "DB_DP".DP[0].Dosi_akt;
      L     #T_Impuls;
      JC    On;
      L     #T_Pause;
On:   T     "DB_DP".DP[0].RestZeit;
      +     -1;
      T     "DB_DP".DP[0].RestZeit;
      JU    Data;

//Handzugabe wird durch Event gefordert
HP:   L     #Restdosierwert;
      T     #Param;
      L     0.0;
      <=R;
      ON    #AUTO;
      AN    #ON;
      R     "DB_DP".DP[0].Meldung;

      AN    "DB_DP".DP[0].Meldung;
      JC    Data;
      R     "DB_DP".DP[0].Meldung;

      L     #count;
      T     #DP_Nr;
      L     "DB_DP".DP[0].LaZa_Nr;
      T     #LZ_NR;

Data: L     #Adr_PC_DB;
      LAR1;
      OPN   "DB_Panel_DP";
      A     #Hand;
      =     DBX [AR1, P#6.5];  //"DB_PC_DP".DoPu[1].Hand
      A     #Kali_Start;
      =     DBX [AR1, P#7.0];  //"DB_PC_DP".DoPu[1].Kali_Start
      A     #Kali_Stop;
      =     DBX [AR1, P#7.1];  //"DB_PC_DP".DoPu[1].Kali_Stop
      A     #DP_An;
      =     DBX [AR1, P#6.6];  //"DB_PC_DP".DoPu[1].ON
      A     #Stoerung;
      =     DBX [AR1, P#6.7];  //"DB_PC_DP".DoPu[1].STM
      L     #Kali_Count;
      T     DBD [AR1, P#36.0];  //"DB_PC_DP".DoPu[1].Kali_Count

      L     #Handzugabe;
      T     DBD [AR1, P#12.0];  //"DB_PC_DP".DoPu[1].Handzugabe
      L     #Restdosierwert;
      T     DBD [AR1, P#20.0];  //"DB_PC_DP".DoPu[1].RestDosierWert

      JU    nexP;
END_FUNCTION

FUNCTION "FC_Blk_Move" : Void   // FC10, STL
{ S7_Optimized_Access := 'FALSE' }
// stored: AutoNumber false
   VAR_INPUT
      Quelle : Int;   // Quelladresse
      Ziel : Int;   // Zieladresse
      Laenge : Int;   // Anzahl zu kopierende Bytes
      _InputBlockDB : DB_ANY;
   END_VAR
   VAR_TEMP
      cntCopy : Int;
      cntToCopy : Int;
      rck : Bool;
      savAr1 : DWord;
      savAr2 : DWord;
   END_VAR
BEGIN

NETWORK
TITLE = 
      OPN   #_InputBlockDB;
// --------------------------------
// Register retten
// --------------------------------
      TAR1;
      T     #savAr1;
      TAR2;
      T     #savAr2;

// --------------------------------
// DW-, W- oder B-Zugriff ermitteln
// --------------------------------
      L     #Quelle;
      L     #Ziel;
      >I;
      JC    sub;
      CAC;
sub:  -I;
      L     4;
      >I;
      JC    set;
      CAC;
set:  T     #cntCopy;
      L     0;
      ==I;
      JC    raus;

// --------------------------------
// Start-Adressen ermitteln
// --------------------------------
      L     #Quelle;
      SLD   3;
      LAR1;

      L     #Ziel;
      SLD   3;
      LAR2;

// --------------------------------
// Kopierrichtung ermitteln
// --------------------------------
      L     #Quelle;
      L     #Ziel;
      <I;
      =     #rck;
      JCN   strL;
      L     #Laenge;
      SLD   3;
      +AR1;
      +AR2;

// --------------------------------
// Daten kopieren
// --------------------------------
strL: L     #Laenge;
retL: T     #cntToCopy;
      L     0;
      <=I;
      JC    raus;
      L     #cntToCopy;
      L     #cntCopy;
      >=I;
      JC    splK;
      CAC;
splK: PUSH;
      AN    #rck;
      JC    splL;
      SLD   3;
      NEGD;
      +AR1;
      +AR2;
splL: POP;
      JL    endL;
      JU    endL;
      JU    byte;
      JU    word;
      JU    tri;
      JU    dwrd;
endL: JU    raus;

byte: L     DBB [AR1, P#0.0];
      T     DBB [AR2, P#0.0];
      JU    nexL;

word: L     DBW [AR1, P#0.0];
      T     DBW [AR2, P#0.0];
      JU    nexL;

tri:  L     DBW [AR1, P#0.0];
      T     DBW [AR2, P#0.0];
      L     DBB [AR1, P#2.0];
      T     DBB [AR2, P#2.0];
      JU    nexL;

dwrd: L     DBD [AR1, P#0.0];
      T     DBD [AR2, P#0.0];
      JU    nexL;

// --------------------------------
// nächter Datenblock
// --------------------------------
nexL: A     #rck;
      JC    subL;
      L     #cntCopy;
      SLD   3;
      +AR1;
      +AR2;
subL: L     #cntToCopy;
      L     #cntCopy;
      -I;
      JU    retL;

// --------------------------------
// Register wiederherstellen
// --------------------------------
raus: L     #savAr1;
      LAR1;
      L     #savAr2;
      LAR2;

END_FUNCTION

FUNCTION "Peripherie" : Void   // FC1090, LAD
TITLE = Anlagenperipherie
{ S7_Optimized_Access := 'TRUE' }
// stored: AutoNumber false, SetENOAutomatically true
   VAR CONSTANT
      Ventilator_aus : Int := 10;
      AUS : USInt;
      Hand_EIN : USInt := 1;
      Hand_AUS : USInt := 2;
      Auto_EIN : USInt := 3;
      Auto_AUS : USInt := 4;
      STOERUNG : USInt := 5;
   END_VAR
BEGIN

REGION Network 1 (SCL): Diverses
   // Deckel Säurebecken
   "Deckel_CM01"();
   "Deckel_CM02"();
   // Schnelllauftor
   "Tor"();
END_REGION

REGION Network 2 (SCL): Sperrluftventilator
   // Frequenzumrichter [7]
   //Ansteuerung
   "Panel".Ventilator.laeuft := ("Panel".Ventilator.Auto OR "Panel".Ventilator.Ein)
   AND "DB_PNOZ_IN_Out".In.PNOZ_OK AND "DB_PNOZ_IN_Out".In.Abluft_ok AND "FU_In_Out".FU[7].PE.Statusbyte.Bereit;

   IF "Panel".Ventilator.laeuft THEN
       "A_Frg_FU_Vent" := TRUE;
   ELSIF "Panel".Ventilator.speed < #Ventilator_aus THEN
       "A_Frg_FU_Vent" := FALSE;
   END_IF;

   "FU_In_Out".FU[7].PA.Steuerwort.FrgHalt := "A_Frg_FU_Vent";
   "FU_In_Out".FU[7].PA.Steuerwort.FrgStop := "A_Frg_FU_Vent";
   "FU_In_Out".FU[7].PA.Steuerwort.RegSp := NOT "FU_In_Out".FU[7].PA.Steuerwort.FrgHalt;

   // Geschwindigkeitsvorgabe
   IF "Panel".Ventilator.laeuft THEN
       IF "Panel".Ventilator.Ein THEN
           "FU_In_Out".FU[7].PA.Speed := "Panel".Ventilator.SW_Hand * 150;
       ELSE
           IF "Uhrzeit".AZ_aktiv THEN
               "FU_In_Out".FU[7].PA.Speed := "Panel".Ventilator.SW_Auto_AZ * 150;
           ELSE
               "FU_In_Out".FU[7].PA.Speed := "Panel".Ventilator.SW_Auto_aAZ * 150;
           END_IF;
       END_IF;
   ELSE
       "FU_In_Out".FU[7].PA.Speed := 0;
   END_IF;

   // --> Panel
   "Panel".Ventilator.betriebsbereit:= "FU_In_Out".FU[7].PE.Statusbyte.Bereit;
   "Panel".Ventilator.Stoerung := "FU_In_Out".FU[7].PE.Statusbyte.Stoer;
   // SEW: 100% == 3000 U/min == 15000 Digits
   "Panel".Ventilator.speed := "FU_In_Out".FU[7].PE.Speed / 150; // in [%]

   "Status_E0A"(Hand:= "Panel".Ventilator.Ein,
                Auto:= "Panel".Ventilator.Auto,
                SonderModus_PumpeSpuelen:=FALSE,
                Stoerung:="FU_In_Out".FU[7].PE.Statusbyte.Stoer OR NOT "FU_In_Out".FU[7].PE.Statusbyte.Bereit,
                Ausgang:= "A_Frg_FU_Vent",
                StatusByte=> "Panel".Ventilator.Status);
END_REGION

REGION Network 3 (SCL): Pumpen
   // Filterpumpen Säure
   "FP_CM01.GP01"();
   "FP_CM02.GP04"();

   // Umwälzpumpen Säure
   "UP_CM01.GP02"();
   "UP_CM02.GP05"();

   // Umwälzpumpen Spüle
   "UP_CM03.GP03"();
   "UP_CM04.GP06"();

   // Versorgung GP13 / GP10
   "Pu_GP01.GP13"();
   "Pu_GP02.GP10"();

   // Entleeren Ver-/Entsorgung GP12 / GP07
   "Pu_GP01.GP12"();
   "Pu_GP02.GP07"();

   // Entleeren Pumpensümpfe GP08 / GP09
   "Pu_CL01.GP08"();
   "Pu_CL02.GP09"();

   // Pumpe GP11 Entleeren Behälter CM05
   "Pu_CM05.GP11_DB"();

   // Status Ventile
   "Ventil_Stati_DB"();
END_REGION

REGION Network 4 (SCL): Pumpe GP14 Entleeren Becken CM01..CM04
   // entsprechende Ventile / Kugelhähne müssen per Hand geöffnet werden
   // Verriegelung mit Max-Niveau Behälter CM05
   // nur Handbetrieb
   "A_CM05.GP14" := "Panel".Pu_Entleeren.Ein AND NOT "E_Niv_max_CM05.BL01";
   // Pumpe Ausschalten
   IF "E_Niv_max_CM05.BL01" THEN
       "Panel".Pu_Entleeren.Ein := FALSE;
   END_IF;
   // --> Visu
   IF "A_CM05.GP14" THEN
       "Panel".Pu_Entleeren.Status := #Hand_EIN;
   ELSE
       "Panel".Pu_Entleeren.Status := #AUS;
   END_IF;
END_REGION
END_FUNCTION

FUNCTION_BLOCK "Deckel"   // FB1190, LAD
TITLE = Deckelsteuerung
{ S7_Optimized_Access := 'TRUE' }
// stored: AutoNumber false, MemoryReserve 100, SetENOAutomatically true
   VAR
      In { ExternalAccessible := 'False'; ExternalVisible := 'False'; ExternalWritable := 'False'} : Struct
         NotHalt : Bool;
         Si_24VDC_links : Bool;
         Si_24VDC_rechts : Bool;
         Auto : Bool;
         Hand : Bool;
         Tipp : Bool;
         ErrQ : Bool;
         T_links_auf : Bool;   // Paneltaste
         T_links_zu : Bool;   // Paneltaste
         T_rechts_auf : Bool;   // Paneltaste
         T_rechts_zu : Bool;   // Paneltaste
         SRM_links_auf : Bool;
         SRM_links_zu : Bool;
         SRM_rechts_auf : Bool;
         SRM_rechts_zu : Bool;
         S_links_auf : Bool;
         S_links_zu : Bool;
         S_rechts_auf : Bool;
         S_rechts_zu : Bool;
      END_STRUCT;
   END_VAR
   VAR RETAIN
      Param { ExternalAccessible := 'False'; ExternalVisible := 'False'; ExternalWritable := 'False'} : Struct
         "TO" : Time := T#27s;
         gleichzeitig : Time := T#1s500ms;
      END_STRUCT;
      Zst { ExternalAccessible := 'False'; ExternalVisible := 'False'; ExternalWritable := 'False'} : Struct
         Fehler : Bool;
         Sperre_Pos_li : Bool;
         Sperre_Pos_re : Bool;
         Req_links_auf : Bool;
         Req_rechts_auf : Bool;
         TW_sicher : Bool;
         Ist_Pos_links : Int;   // 0% = auf; 100% = zu
         Ist_Pos_rechts : Int;   // 0% = auf; 100% = zu
      END_STRUCT;
      Out { ExternalAccessible := 'False'; ExternalVisible := 'False'; ExternalWritable := 'False'} : Struct
         links_auf : Bool;
         links_zu : Bool;
         rechts_auf : Bool;
         rechts_zu : Bool;
      END_STRUCT;
      Mld { ExternalAccessible := 'False'; ExternalVisible := 'False'; ExternalWritable := 'False'} : Struct
         TO_links_auf : Bool;
         TO_links_zu : Bool;
         TO_rechts_auf : Bool;
         TO_rechts_zu : Bool;
         Si_24VDC_links : Bool;
         Si_24VDC_rechts : Bool;
         n_Auto : Bool;
         SF_gleich_li_auf : Bool;
         SF_gleich_li_zu : Bool;
         SF_gleich_re_auf : Bool;
         SF_gleich_re_zu : Bool;
      END_STRUCT;
   END_VAR
   VAR
      IEC_Timer { ExternalAccessible := 'False'; ExternalVisible := 'False'; ExternalWritable := 'False'} : Struct
         TO_li_auf { S7_SetPoint := 'True'} : TON_TIME;
         TO_li_zu { S7_SetPoint := 'True'} : TON_TIME;
         TO_re_auf { S7_SetPoint := 'True'} : TON_TIME;
         TO_re_zu { S7_SetPoint := 'True'} : TON_TIME;
         gleich_li_auf { S7_SetPoint := 'True'} : TON_TIME;
         gleich_li_zu { S7_SetPoint := 'True'} : TON_TIME;
         gleich_re_auf { S7_SetPoint := 'True'} : TON_TIME;
         gleich_re_zu { S7_SetPoint := 'True'} : TON_TIME;
      END_STRUCT;
   END_VAR
   VAR_TEMP
      TO_links_auf : Bool;
      TO_links_zu : Bool;
      TO_rechts_auf : Bool;
      TO_rechts_zu : Bool;
   END_VAR
BEGIN

REGION Network 1 (SCL): Input / Sammelstörung
   // Panelbedienung und Sensoren --> Input()
   // Not-Halt
   #In.NotHalt :=  NOT "DB_PNOZ_IN_Out".In.NH_Frg_Deckel;

   IF #In.ErrQ THEN
       #Zst.Fehler := FALSE;
   END_IF;

   IF #In.NotHalt OR NOT #In.Si_24VDC_links OR NOT #In.Si_24VDC_rechts OR #Mld.TO_links_auf OR #Mld.TO_links_zu
       OR #Mld.TO_rechts_auf OR #Mld.TO_rechts_zu
   THEN
       #Zst.Fehler := TRUE;
   END_IF;
END_REGION

REGION Network 2 (SCL): Ansteuerung
   IF NOT #Zst.Fehler THEN
       IF #In.Auto AND #Zst.TW_sicher THEN // Automatikbetrieb
           // Linke Seite
           #Out.links_auf := #Zst.Req_links_auf;
           #Out.links_zu := NOT #Zst.Req_links_auf;
           // Rechte Seite
           #Out.rechts_auf := #Zst.Req_rechts_auf;
           #Out.rechts_zu := NOT #Zst.Req_rechts_auf;

       ELSIF #In.Hand AND #Zst.TW_sicher THEN // Handbetrieb
           // Linke Seite
           IF #In.T_links_auf AND NOT #In.T_links_zu THEN
               #Out.links_auf := TRUE;
               #Out.links_zu := FALSE;
           END_IF;
           IF #In.T_links_zu AND NOT #In.T_links_auf THEN
               #Out.links_zu := TRUE;
               #Out.links_auf := FALSE;
           END_IF;
           // Rechte Seite
           IF #In.T_rechts_auf AND NOT #In.T_rechts_zu THEN
               #Out.rechts_auf := TRUE;
               #Out.rechts_zu := FALSE;
           END_IF;
           IF #In.T_rechts_zu AND NOT #In.T_rechts_auf THEN
               #Out.rechts_zu := TRUE;
               #Out.rechts_auf := FALSE;
           END_IF;
       ELSIF #In.Tipp THEN  // Tippbetrieb
           // Linke Seite
           #Out.links_auf := #In.T_links_auf AND NOT #In.T_links_zu;
           #Out.links_zu := #In.T_links_zu AND NOT #In.T_links_auf AND #Zst.TW_sicher;

           // Rechte Seite
           #Out.rechts_auf := #In.T_rechts_auf AND NOT #In.T_rechts_zu;
           #Out.rechts_zu := #In.T_rechts_zu AND NOT #In.T_rechts_auf AND #Zst.TW_sicher;
       ELSE
           #Out.links_auf := FALSE;
           #Out.links_zu := FALSE;
           #Out.rechts_auf := FALSE;
           #Out.rechts_zu := FALSE;
       END_IF;

   ELSE // Not-Halt
       #Out.links_auf := FALSE;
       #Out.links_zu := FALSE;
       #Out.rechts_auf := FALSE;
       #Out.rechts_zu := FALSE;
   END_IF;

   // Endlagen erreicht
   IF #In.S_links_auf OR #In.SRM_links_auf THEN
       #Out.links_auf := FALSE;
   END_IF;
   IF #In.S_links_zu OR #In.SRM_links_zu THEN
       #Out.links_zu := FALSE;
   END_IF;
   IF #In.S_rechts_auf OR #In.SRM_rechts_auf THEN
       #Out.rechts_auf := FALSE;
   END_IF;
   IF #In.S_rechts_zu OR #In.SRM_rechts_zu THEN
       #Out.rechts_zu := FALSE;
   END_IF;


   REGION Ist-Position
       // Ist-Pos simulieren für Visu 
       IF #Out.links_auf AND "Imp_10Hz" AND NOT #In.S_links_auf THEN
           #Zst.Ist_Pos_links := MAX(IN1 := 5, IN2 := (#Zst.Ist_Pos_links - 1));
       ELSIF #In.S_links_auf THEN
           #Zst.Ist_Pos_links := 0;
       END_IF;

       IF #Out.rechts_auf AND "Imp_10Hz" AND NOT #In.S_rechts_auf THEN
           #Zst.Ist_Pos_rechts := MAX(IN1 := 5, IN2 := (#Zst.Ist_Pos_rechts - 1));
       ELSIF #In.S_rechts_auf THEN
           #Zst.Ist_Pos_rechts := 0;
       END_IF;

       // Ist-Pos simulieren für Visu 
       IF #Out.links_zu AND "Imp_5Hz" AND NOT #In.S_links_zu THEN
           #Zst.Ist_Pos_links := MIN(IN1 := 95, IN2 := (#Zst.Ist_Pos_links + 1));
       ELSIF #In.S_links_zu THEN
           #Zst.Ist_Pos_links := 100;
       END_IF;

       IF #Out.rechts_zu AND "Imp_5Hz" AND NOT #In.S_rechts_zu THEN
           #Zst.Ist_Pos_rechts := MIN(IN1 := 95, IN2 := (#Zst.Ist_Pos_rechts + 1));
       ELSIF #In.S_rechts_zu THEN
           #Zst.Ist_Pos_rechts := 100;
       END_IF;
   END_REGION
END_REGION

REGION Network 3 (SCL): Possperre
   // Überfahren verboten
   #Zst.Sperre_Pos_li := NOT (#In.S_links_auf XOR #In.S_links_zu)  OR #Out.links_auf OR #Out.links_zu;

   #Zst.Sperre_Pos_re := NOT (#In.S_rechts_auf XOR #In.S_rechts_zu) OR #Out.rechts_auf OR #Out.rechts_zu;
END_REGION

REGION Network 4 (SCL): Überwachung / Alarme
   // Sicherungsfall / Zeitüberschreitung
   // Sicherungsfall 24V DC links
   #Mld.Si_24VDC_links := NOT #In.Si_24VDC_links AND NOT #In.NotHalt;
   // Sicherungsfall 24V DC rechts
   #Mld.Si_24VDC_rechts := NOT #In.Si_24VDC_rechts AND NOT #In.NotHalt;

